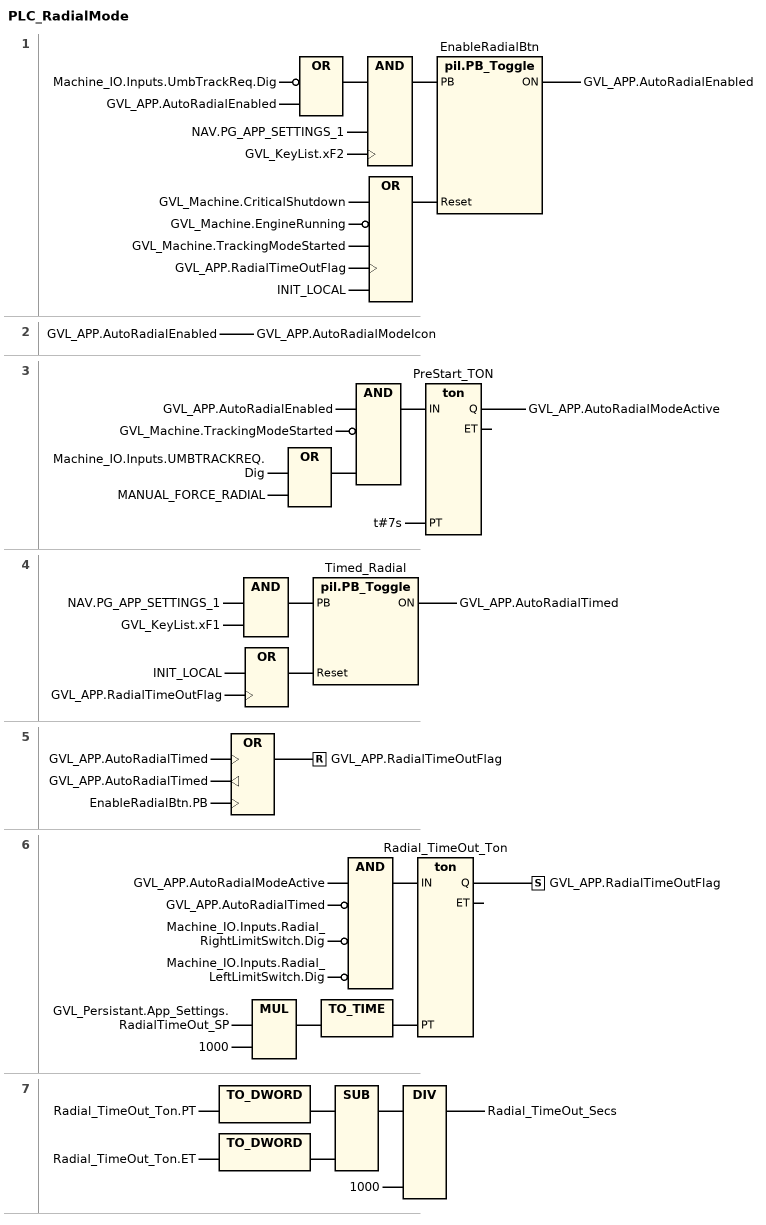
// NETWORK 1
_rt1(CLK := GVL_KeyList.xF2);
_rt2(CLK := GVL_APP.RadialTimeOutFlag);
EnableRadialBtn(PB := (NOT Machine_IO.Inputs.UmbTrackReq.Dig OR GVL_APP.AutoRadialEnabled) AND NAV.PG_APP_SETTINGS_1 AND _rt1.Q, Reset := GVL_Machine.CriticalShutdown OR NOT GVL_Machine.EngineRunning OR GVL_Machine.TrackingModeStarted OR _rt2.Q OR INIT_LOCAL); // pil.PB_Toggle
GVL_APP.AutoRadialEnabled := EnableRadialBtn.ON;

// NETWORK 2
GVL_APP.AutoRadialModeIcon := GVL_APP.AutoRadialEnabled;

// NETWORK 3
PreStart_TON(IN := GVL_APP.AutoRadialEnabled AND NOT GVL_Machine.TrackingModeStarted AND (Machine_IO.Inputs.UMBTRACKREQ.Dig OR MANUAL_FORCE_RADIAL), PT := t#7s); // ton
GVL_APP.AutoRadialModeActive := PreStart_TON.Q;

// NETWORK 4
_rt3(CLK := GVL_APP.RadialTimeOutFlag);
Timed_Radial(PB := NAV.PG_APP_SETTINGS_1 AND GVL_KeyList.xF1, Reset := INIT_LOCAL OR _rt3.Q); // pil.PB_Toggle
GVL_APP.AutoRadialTimed := Timed_Radial.ON;

// NETWORK 5
_rt4(CLK := GVL_APP.AutoRadialTimed);
_ft1(CLK := GVL_APP.AutoRadialTimed);
_rt5(CLK := EnableRadialBtn.PB);
GVL_APP.RadialTimeOutFlag R= _rt4.Q OR _ft1.Q OR _rt5.Q;

// NETWORK 6
Radial_TimeOut_Ton(IN := GVL_APP.AutoRadialModeActive AND NOT GVL_APP.AutoRadialTimed AND NOT Machine_IO.Inputs.Radial_RightLimitSwitch.Dig AND NOT Machine_IO.Inputs.Radial_LeftLimitSwitch.Dig, PT := TO_TIME(GVL_Persistant.App_Settings.RadialTimeOut_SP * 1000)); // ton
GVL_APP.RadialTimeOutFlag S= Radial_TimeOut_Ton.Q;

// NETWORK 7
Radial_TimeOut_Secs := (TO_DWORD(Radial_TimeOut_Ton.PT) - TO_DWORD(Radial_TimeOut_Ton.ET)) / 1000;

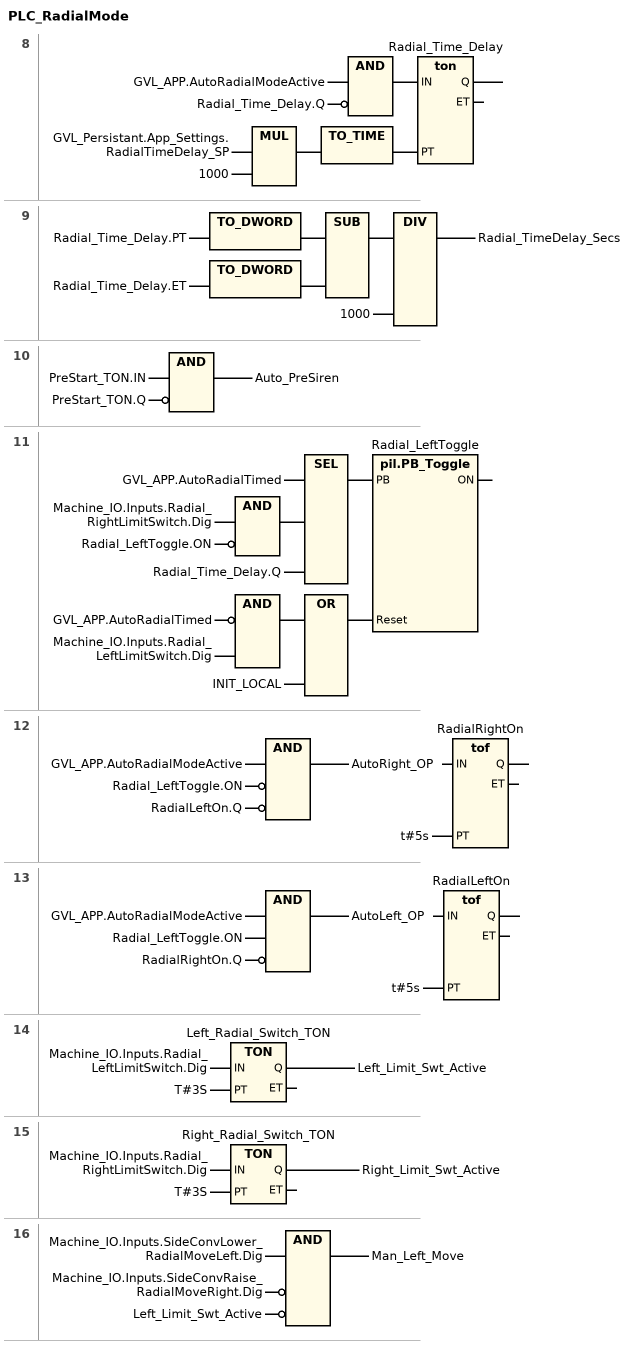
// NETWORK 8
Radial_Time_Delay(IN := GVL_APP.AutoRadialModeActive AND NOT Radial_Time_Delay.Q, PT := TO_TIME(GVL_Persistant.App_Settings.RadialTimeDelay_SP * 1000)); // ton

// NETWORK 9
Radial_TimeDelay_Secs := (TO_DWORD(Radial_Time_Delay.PT) - TO_DWORD(Radial_Time_Delay.ET)) / 1000;

// NETWORK 10
Auto_PreSiren := PreStart_TON.IN AND NOT PreStart_TON.Q;

// NETWORK 11
Radial_LeftToggle(PB := SEL(GVL_APP.AutoRadialTimed, Machine_IO.Inputs.Radial_RightLimitSwitch.Dig AND NOT Radial_LeftToggle.ON, Radial_Time_Delay.Q), Reset := NOT GVL_APP.AutoRadialTimed AND Machine_IO.Inputs.Radial_LeftLimitSwitch.Dig OR INIT_LOCAL); // pil.PB_Toggle

// NETWORK 12
_w1 := GVL_APP.AutoRadialModeActive AND NOT Radial_LeftToggle.ON AND NOT RadialLeftOn.Q;
AutoRight_OP := _w1;
RadialRightOn(IN := _w1, PT := t#5s); // tof

// NETWORK 13
_w2 := GVL_APP.AutoRadialModeActive AND Radial_LeftToggle.ON AND NOT RadialRightOn.Q;
AutoLeft_OP := _w2;
RadialLeftOn(IN := _w2, PT := t#5s); // tof

// NETWORK 14
Left_Radial_Switch_TON(IN := Machine_IO.Inputs.Radial_LeftLimitSwitch.Dig, PT := T#3S); // TON
Left_Limit_Swt_Active := Left_Radial_Switch_TON.Q;

// NETWORK 15
Right_Radial_Switch_TON(IN := Machine_IO.Inputs.Radial_RightLimitSwitch.Dig, PT := T#3S); // TON
Right_Limit_Swt_Active := Right_Radial_Switch_TON.Q;

// NETWORK 16
Man_Left_Move := Machine_IO.Inputs.SideConvLower_RadialMoveLeft.Dig AND NOT Machine_IO.Inputs.SideConvRaise_RadialMoveRight.Dig AND NOT Left_Limit_Swt_Active;

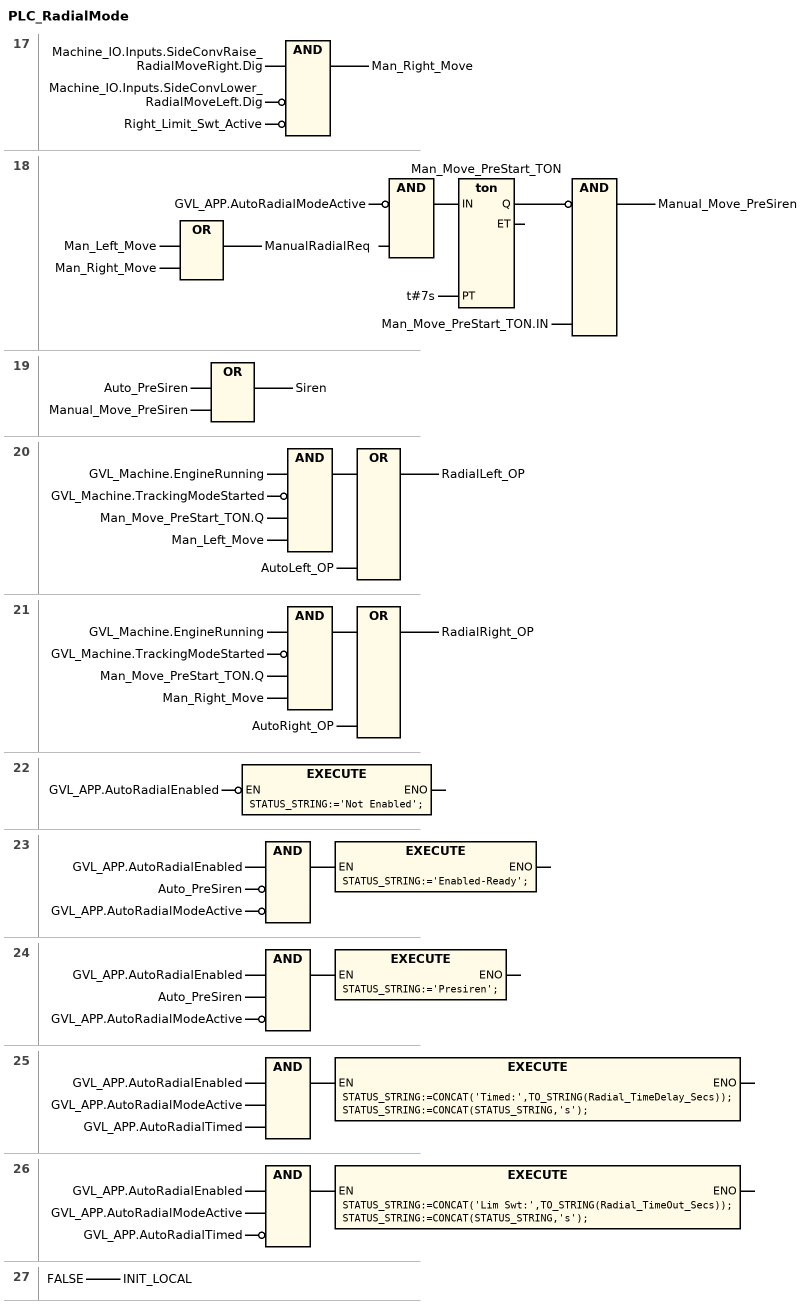
// NETWORK 17
Man_Right_Move := Machine_IO.Inputs.SideConvRaise_RadialMoveRight.Dig AND NOT Machine_IO.Inputs.SideConvLower_RadialMoveLeft.Dig AND NOT Right_Limit_Swt_Active;

// NETWORK 18
_w3 := Man_Left_Move OR Man_Right_Move;
ManualRadialReq := _w3;
Man_Move_PreStart_TON(IN := NOT GVL_APP.AutoRadialModeActive AND _w3, PT := t#7s); // ton
Manual_Move_PreSiren := NOT Man_Move_PreStart_TON.Q AND Man_Move_PreStart_TON.IN;

// NETWORK 19
Siren := Auto_PreSiren OR Manual_Move_PreSiren;

// NETWORK 20
RadialLeft_OP := GVL_Machine.EngineRunning AND NOT GVL_Machine.TrackingModeStarted AND Man_Move_PreStart_TON.Q AND Man_Left_Move OR AutoLeft_OP;

// NETWORK 21
RadialRight_OP := GVL_Machine.EngineRunning AND NOT GVL_Machine.TrackingModeStarted AND Man_Move_PreStart_TON.Q AND Man_Right_Move OR AutoRight_OP;

// NETWORK 22
IF NOT GVL_APP.AutoRadialEnabled THEN STATUS_STRING:='Not Enabled'; END_IF

// NETWORK 23
IF GVL_APP.AutoRadialEnabled AND NOT Auto_PreSiren AND NOT GVL_APP.AutoRadialModeActive THEN
    STATUS_STRING:='Enabled-Ready';
END_IF

// NETWORK 24
IF GVL_APP.AutoRadialEnabled AND Auto_PreSiren AND NOT GVL_APP.AutoRadialModeActive THEN
    STATUS_STRING:='Presiren';
END_IF

// NETWORK 25
IF GVL_APP.AutoRadialEnabled AND GVL_APP.AutoRadialModeActive AND GVL_APP.AutoRadialTimed THEN
    STATUS_STRING:=CONCAT('Timed:',TO_STRING(Radial_TimeDelay_Secs));
    STATUS_STRING:=CONCAT(STATUS_STRING,'s');
END_IF

// NETWORK 26
IF GVL_APP.AutoRadialEnabled AND GVL_APP.AutoRadialModeActive AND NOT GVL_APP.AutoRadialTimed THEN
    STATUS_STRING:=CONCAT('Lim Swt:',TO_STRING(Radial_TimeOut_Secs));
    STATUS_STRING:=CONCAT(STATUS_STRING,'s');
END_IF

// NETWORK 27
INIT_LOCAL := FALSE;

END_PROGRAM

// Device/Application/App_PLC/Control/PLC_JackLegs_SideConv
PROGRAM PLC_JackLegs_SideConv
VAR
	Prestart_TON: TON;
	Enable: BOOL;
	Siren: BOOL;
	Man_Side_Conv_Raise: BOOL;
	Man_Side_Conv_Lower: BOOL;
	Man_LHS_JackLegRaise: BOOL;
	Man_LHS_JackLegLower: BOOL;
	Man_RHS_JackLegRaise: BOOL;
	Man_RHS_JackLegLower: BOOL;
END_VAR
VAR // added by the converter: edge detectors and wires of the graphical bodies
    _w1 : BOOL;
END_VAR

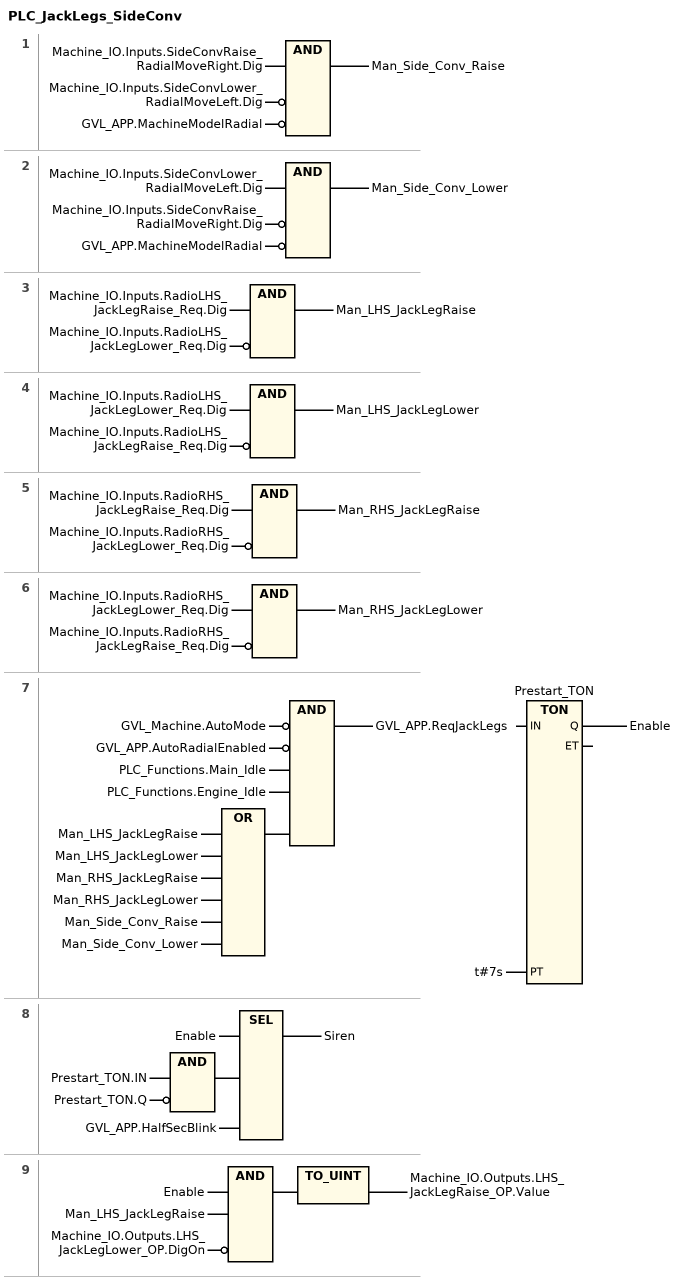
// NETWORK 1
Man_Side_Conv_Raise := Machine_IO.Inputs.SideConvRaise_RadialMoveRight.Dig AND NOT Machine_IO.Inputs.SideConvLower_RadialMoveLeft.Dig AND NOT GVL_APP.MachineModelRadial;

// NETWORK 2
Man_Side_Conv_Lower := Machine_IO.Inputs.SideConvLower_RadialMoveLeft.Dig AND NOT Machine_IO.Inputs.SideConvRaise_RadialMoveRight.Dig AND NOT GVL_APP.MachineModelRadial;

// NETWORK 3
Man_LHS_JackLegRaise := Machine_IO.Inputs.RadioLHS_JackLegRaise_Req.Dig AND NOT Machine_IO.Inputs.RadioLHS_JackLegLower_Req.Dig;

// NETWORK 4
Man_LHS_JackLegLower := Machine_IO.Inputs.RadioLHS_JackLegLower_Req.Dig AND NOT Machine_IO.Inputs.RadioLHS_JackLegRaise_Req.Dig;

// NETWORK 5
Man_RHS_JackLegRaise := Machine_IO.Inputs.RadioRHS_JackLegRaise_Req.Dig AND NOT Machine_IO.Inputs.RadioRHS_JackLegLower_Req.Dig;

// NETWORK 6
Man_RHS_JackLegLower := Machine_IO.Inputs.RadioRHS_JackLegLower_Req.Dig AND NOT Machine_IO.Inputs.RadioRHS_JackLegRaise_Req.Dig;

// NETWORK 7
_w1 := NOT GVL_Machine.AutoMode AND NOT GVL_APP.AutoRadialEnabled AND PLC_Functions.Main_Idle AND PLC_Functions.Engine_Idle AND (Man_LHS_JackLegRaise OR Man_LHS_JackLegLower OR Man_RHS_JackLegRaise OR Man_RHS_JackLegLower OR Man_Side_Conv_Raise OR Man_Side_Conv_Lower);
GVL_APP.ReqJackLegs := _w1;
Prestart_TON(IN := _w1, PT := t#7s); // TON
Enable := Prestart_TON.Q;

// NETWORK 8
Siren := SEL(Enable, Prestart_TON.IN AND NOT Prestart_TON.Q, GVL_APP.HalfSecBlink);

// NETWORK 9
Machine_IO.Outputs.LHS_JackLegRaise_OP.Value := TO_UINT(Enable AND Man_LHS_JackLegRaise AND NOT Machine_IO.Outputs.LHS_JackLegLower_OP.DigOn);

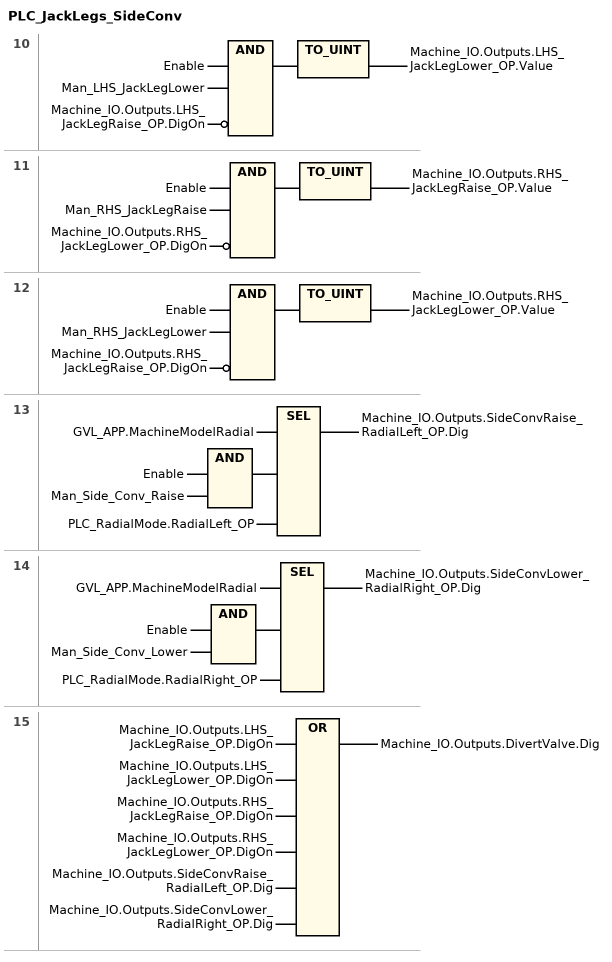
// NETWORK 10
Machine_IO.Outputs.LHS_JackLegLower_OP.Value := TO_UINT(Enable AND Man_LHS_JackLegLower AND NOT Machine_IO.Outputs.LHS_JackLegRaise_OP.DigOn);

// NETWORK 11
Machine_IO.Outputs.RHS_JackLegRaise_OP.Value := TO_UINT(Enable AND Man_RHS_JackLegRaise AND NOT Machine_IO.Outputs.RHS_JackLegLower_OP.DigOn);

// NETWORK 12
Machine_IO.Outputs.RHS_JackLegLower_OP.Value := TO_UINT(Enable AND Man_RHS_JackLegLower AND NOT Machine_IO.Outputs.RHS_JackLegRaise_OP.DigOn);

// NETWORK 13
Machine_IO.Outputs.SideConvRaise_RadialLeft_OP.Dig := SEL(GVL_APP.MachineModelRadial, Enable AND Man_Side_Conv_Raise, PLC_RadialMode.RadialLeft_OP);

// NETWORK 14
Machine_IO.Outputs.SideConvLower_RadialRight_OP.Dig := SEL(GVL_APP.MachineModelRadial, Enable AND Man_Side_Conv_Lower, PLC_RadialMode.RadialRight_OP);

// NETWORK 15
Machine_IO.Outputs.DivertValve.Dig := Machine_IO.Outputs.LHS_JackLegRaise_OP.DigOn OR Machine_IO.Outputs.LHS_JackLegLower_OP.DigOn OR Machine_IO.Outputs.RHS_JackLegRaise_OP.DigOn OR Machine_IO.Outputs.RHS_JackLegLower_OP.DigOn OR Machine_IO.Outputs.SideConvRaise_RadialLeft_OP.Dig OR Machine_IO.Outputs.SideConvLower_RadialRight_OP.Dig;

END_PROGRAM

// Device/Application/App_PLC/PLC_FanCtrl
PROGRAM PLC_FanCtrl
VAR
	OneSecTon: TON;
	Step: BYTE;
	WaitTon1: TON;
	WaitTon2: TON;

	RevTime_sec: WORD;
	THERMOSTAT: BOOL;
	//Fan_Forward_Time_Secs: UINT;
	STATUS_STRING: STRING;
	Forward_Time_Remaining: DWORD;
	Reverse_Time_Remaining: DWORD;
	Current_Forward_Time_STR: STRING;
END_VAR

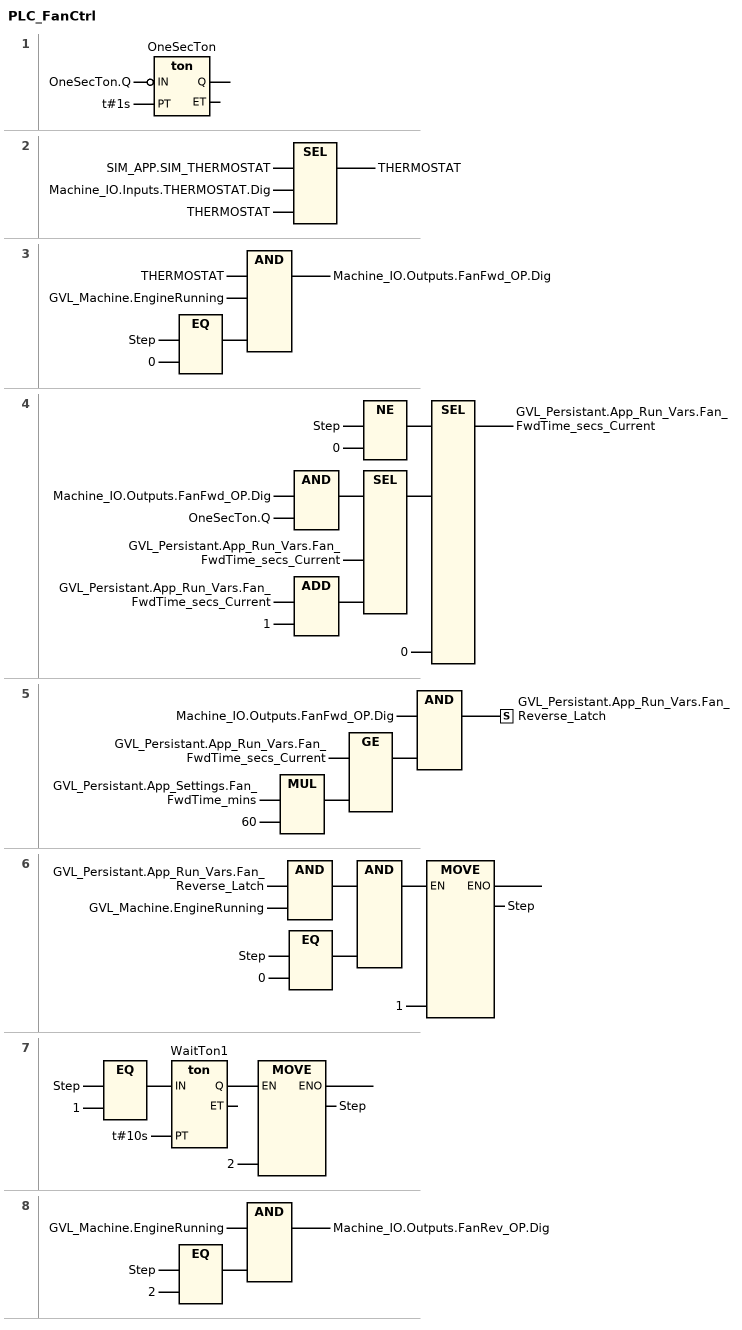
// NETWORK 1
OneSecTon(IN := NOT OneSecTon.Q, PT := t#1s); // ton

// NETWORK 2
THERMOSTAT := SEL(SIM_APP.SIM_THERMOSTAT, Machine_IO.Inputs.THERMOSTAT.Dig, THERMOSTAT);

// NETWORK 3
Machine_IO.Outputs.FanFwd_OP.Dig := THERMOSTAT AND GVL_Machine.EngineRunning AND Step = 0;

// NETWORK 4
GVL_Persistant.App_Run_Vars.Fan_FwdTime_secs_Current := SEL(Step <> 0, SEL(Machine_IO.Outputs.FanFwd_OP.Dig AND OneSecTon.Q, GVL_Persistant.App_Run_Vars.Fan_FwdTime_secs_Current, GVL_Persistant.App_Run_Vars.Fan_FwdTime_secs_Current + 1), 0);

// NETWORK 5
GVL_Persistant.App_Run_Vars.Fan_Reverse_Latch S= Machine_IO.Outputs.FanFwd_OP.Dig AND GVL_Persistant.App_Run_Vars.Fan_FwdTime_secs_Current >= GVL_Persistant.App_Settings.Fan_FwdTime_mins * 60;

// NETWORK 6
IF (GVL_Persistant.App_Run_Vars.Fan_Reverse_Latch AND GVL_Machine.EngineRunning) AND Step = 0 THEN
    Step := 1;
END_IF

// NETWORK 7
WaitTon1(IN := Step = 1, PT := t#10s); // ton
IF WaitTon1.Q THEN Step := 2; END_IF

// NETWORK 8
Machine_IO.Outputs.FanRev_OP.Dig := GVL_Machine.EngineRunning AND Step = 2;

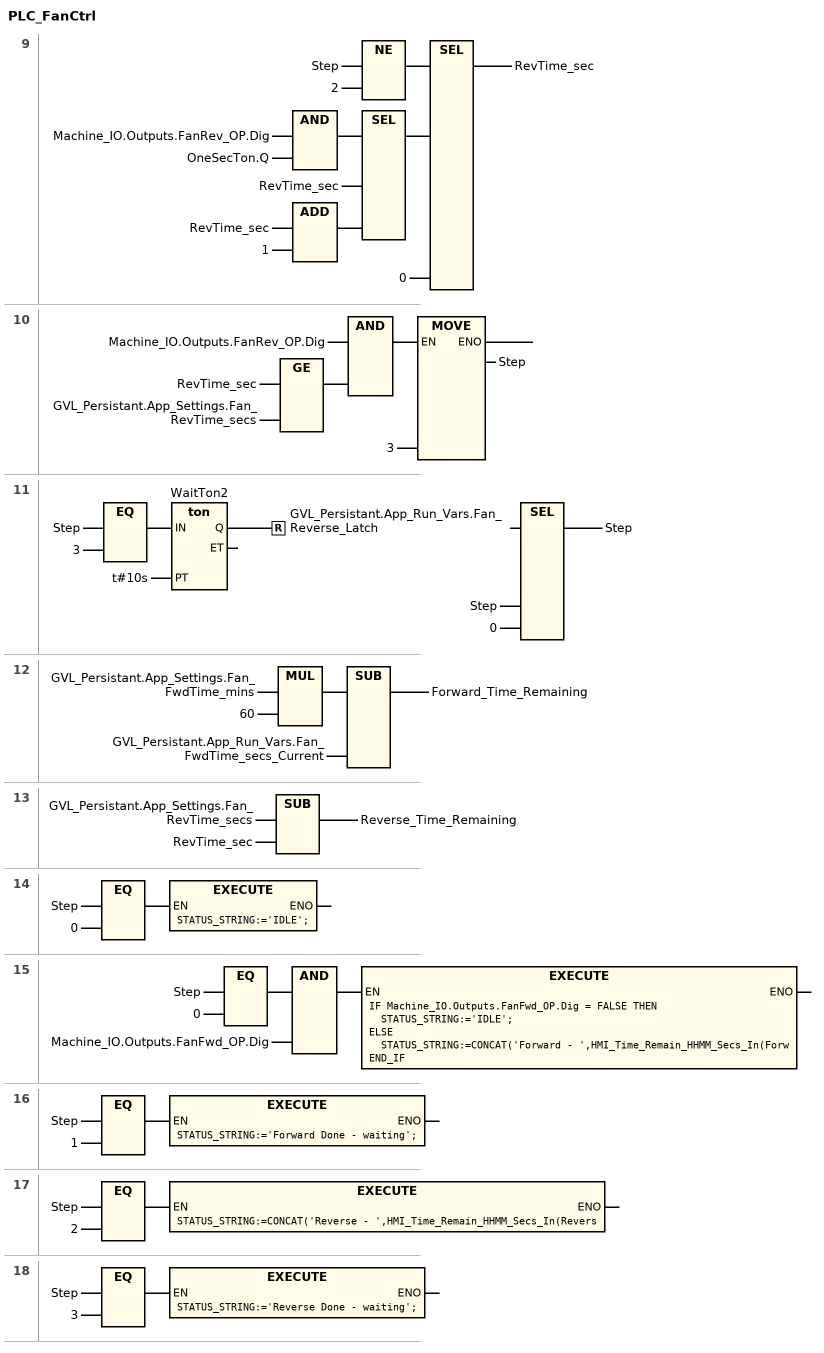
// NETWORK 9
RevTime_sec := SEL(Step <> 2, SEL(Machine_IO.Outputs.FanRev_OP.Dig AND OneSecTon.Q, RevTime_sec, RevTime_sec + 1), 0);

// NETWORK 10
IF Machine_IO.Outputs.FanRev_OP.Dig AND RevTime_sec >= GVL_Persistant.App_Settings.Fan_RevTime_secs THEN
    Step := 3;
END_IF

// NETWORK 11
WaitTon2(IN := Step = 3, PT := t#10s); // ton
GVL_Persistant.App_Run_Vars.Fan_Reverse_Latch R= WaitTon2.Q;
Step := SEL(WaitTon2.Q, Step, 0);

// NETWORK 12
Forward_Time_Remaining := GVL_Persistant.App_Settings.Fan_FwdTime_mins * 60 - GVL_Persistant.App_Run_Vars.Fan_FwdTime_secs_Current;

// NETWORK 13
Reverse_Time_Remaining := GVL_Persistant.App_Settings.Fan_RevTime_secs - RevTime_sec;

// NETWORK 14
IF Step = 0 THEN STATUS_STRING:='IDLE'; END_IF

// NETWORK 15
IF Step = 0 AND Machine_IO.Outputs.FanFwd_OP.Dig THEN
    IF Machine_IO.Outputs.FanFwd_OP.Dig = FALSE THEN
    	STATUS_STRING:='IDLE';
    ELSE
    	STATUS_STRING:=CONCAT('Forward - ',HMI_Time_Remain_HHMM_Secs_In(Forward_Time_Remaining));	
    END_IF
END_IF

// NETWORK 16
IF Step = 1 THEN STATUS_STRING:='Forward Done - waiting'; END_IF

// NETWORK 17
IF Step = 2 THEN STATUS_STRING:=CONCAT('Reverse - ',HMI_Time_Remain_HHMM_Secs_In(Reverse_Time_Remaining)); END_IF

// NETWORK 18
IF Step = 3 THEN STATUS_STRING:='Reverse Done - waiting'; END_IF

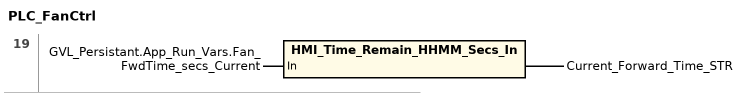
// NETWORK 19
Current_Forward_Time_STR := HMI_Time_Remain_HHMM_Secs_In(In := GVL_Persistant.App_Run_Vars.Fan_FwdTime_secs_Current);

END_PROGRAM

// Device/Application/App_PLC/CAN Comms/Engine Comms/HMI_Time_Remain_HHMM_Secs_In
FUNCTION HMI_Time_Remain_HHMM_Secs_In : STRING
VAR_INPUT
	In:DWORD;
END_VAR
VAR
	TotalSeconds: DWORD;
	Hours: DWORD;
	Mins: DWORD;
	Secs: DWORD;
	
	Temp_STR:STRING;
	TotalMinutes: DWORD;
END_VAR

TotalSeconds:=TO_DWORD(In);

TotalMinutes:=(TotalSeconds MOD (24*60*60))/60;

Hours:=TotalSeconds/(60*60);
Mins:=(TotalSeconds MOD (60*60))/60;
Secs:=TotalSeconds MOD 60;

Temp_STR:= '';

Temp_STR:= CONCAT(Temp_STR,DWORD_TO_STRING(Hours));
IF Hours < 10 THEN
	Temp_STR:= CONCAT(Temp_STR,'0');
END_IF

Temp_STR:= CONCAT(Temp_STR,':');

IF Mins < 10 THEN
	Temp_STR:= CONCAT(Temp_STR,'0');
END_IF
Temp_STR:= CONCAT(Temp_STR,DWORD_TO_STRING(Mins));

Temp_STR:= CONCAT(Temp_STR,':');

IF Secs < 10 THEN
	Temp_STR:= CONCAT(Temp_STR,'0');
END_IF
Temp_STR:= CONCAT(Temp_STR,DWORD_TO_STRING(Secs));


HMI_Time_Remain_HHMM_Secs_In := Temp_STR;

END_FUNCTION

// Device/Application/App_PLC/PLC_EngineRun
PROGRAM PLC_EngineRun
VAR
	TestBit1: BOOL;
	TempWord: WORD;
	TOF_0: tof;

	PreSirenTrig: BOOL;
	PreSirenTon: ton;
	PreSiren: BOOL;
	
	FastBlinkWait: ton;
	FastCountBlink: blink;
	FastBlinkTrig: R_trig;
	EngineSpeedPos_Count: SP_Count_VAR;
	
	WaitTon1: ton;
	WaitTof1: tof;

	TON_0: ton;
	BLINK_0: blink;
	PwrUpReset: BOOL;
	ECU_ENABLE: BOOL;
	SR_Auto_Stopped: SR;
END_VAR
VAR // added by the converter: edge detectors and wires of the graphical bodies
    _w1 : BOOL;
    _rt1, _rt2, _rt3 : R_TRIG;
    _ft1 : F_TRIG;
END_VAR

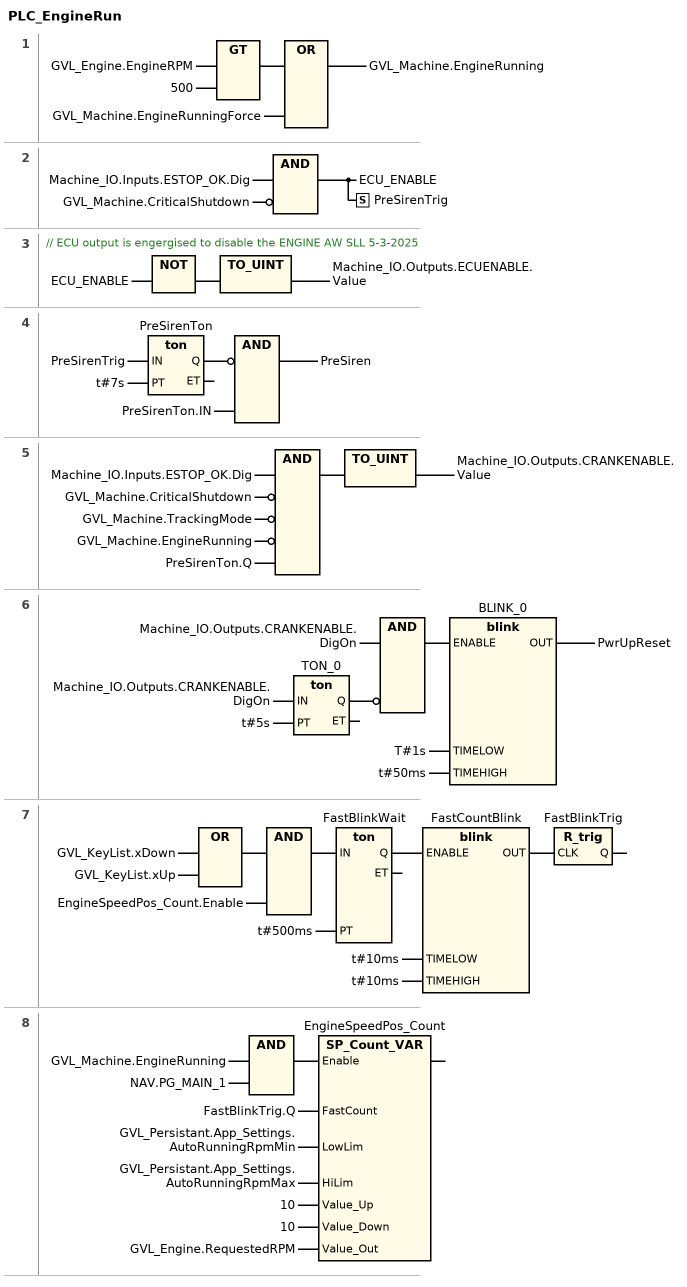
// NETWORK 1
GVL_Machine.EngineRunning := GVL_Engine.EngineRPM > 500 OR GVL_Machine.EngineRunningForce;

// NETWORK 2
_w1 := Machine_IO.Inputs.ESTOP_OK.Dig AND NOT GVL_Machine.CriticalShutdown;
ECU_ENABLE := _w1;
PreSirenTrig S= _w1;

// NETWORK 3
// // ECU output is engergised to disable the ENGINE AW SLL 5-3-2025
Machine_IO.Outputs.ECUENABLE.Value := TO_UINT(NOT ECU_ENABLE);

// NETWORK 4
PreSirenTon(IN := PreSirenTrig, PT := t#7s); // ton
PreSiren := NOT PreSirenTon.Q AND PreSirenTon.IN;

// NETWORK 5
Machine_IO.Outputs.CRANKENABLE.Value := TO_UINT(Machine_IO.Inputs.ESTOP_OK.Dig AND NOT GVL_Machine.CriticalShutdown AND NOT GVL_Machine.TrackingMode AND NOT GVL_Machine.EngineRunning AND PreSirenTon.Q);

// NETWORK 6
TON_0(IN := Machine_IO.Outputs.CRANKENABLE.DigOn, PT := t#5s); // ton
BLINK_0(ENABLE := Machine_IO.Outputs.CRANKENABLE.DigOn AND NOT TON_0.Q, TIMELOW := T#1s, TIMEHIGH := t#50ms); // blink
PwrUpReset := BLINK_0.OUT;

// NETWORK 7
FastBlinkWait(IN := (GVL_KeyList.xDown OR GVL_KeyList.xUp) AND EngineSpeedPos_Count.Enable, PT := t#500ms); // ton
FastCountBlink(ENABLE := FastBlinkWait.Q, TIMELOW := t#10ms, TIMEHIGH := t#10ms); // blink
FastBlinkTrig(CLK := FastCountBlink.OUT); // R_trig

// NETWORK 8
EngineSpeedPos_Count(
    Enable := GVL_Machine.EngineRunning AND NAV.PG_MAIN_1,
    FastCount := FastBlinkTrig.Q,
    LowLim := GVL_Persistant.App_Settings.AutoRunningRpmMin,
    HiLim := GVL_Persistant.App_Settings.AutoRunningRpmMax,
    Value_Up := 10,
    Value_Down := 10,
    Value_Out := GVL_Engine.RequestedRPM); // SP_Count_VAR

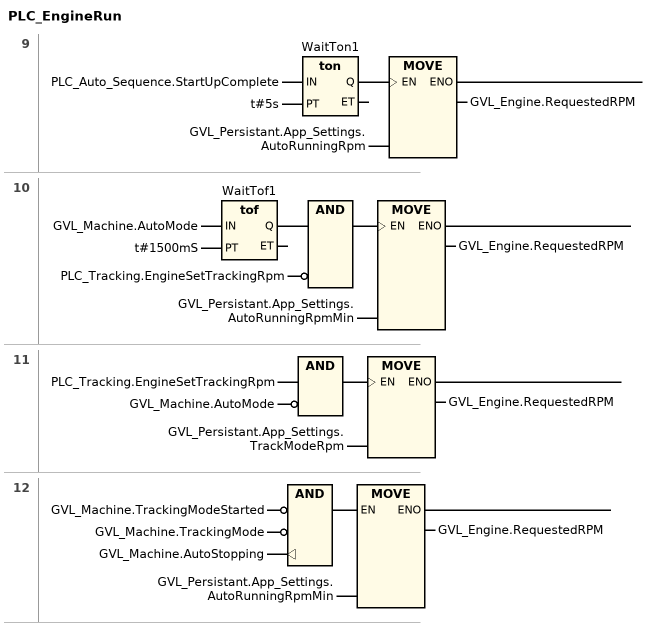
// NETWORK 9
WaitTon1(IN := PLC_Auto_Sequence.StartUpComplete, PT := t#5s); // ton
_rt1(CLK := WaitTon1.Q);
IF _rt1.Q THEN GVL_Engine.RequestedRPM := GVL_Persistant.App_Settings.AutoRunningRpm; END_IF

// NETWORK 10
WaitTof1(IN := GVL_Machine.AutoMode, PT := t#1500mS); // tof
_rt2(CLK := WaitTof1.Q AND NOT PLC_Tracking.EngineSetTrackingRpm);
IF _rt2.Q THEN GVL_Engine.RequestedRPM := GVL_Persistant.App_Settings.AutoRunningRpmMin; END_IF

// NETWORK 11
_rt3(CLK := PLC_Tracking.EngineSetTrackingRpm AND NOT GVL_Machine.AutoMode);
IF _rt3.Q THEN GVL_Engine.RequestedRPM := GVL_Persistant.App_Settings.TrackModeRpm; END_IF

// NETWORK 12
_ft1(CLK := GVL_Machine.AutoStopping);
IF NOT GVL_Machine.TrackingModeStarted AND NOT GVL_Machine.TrackingMode AND _ft1.Q THEN
    GVL_Engine.RequestedRPM := GVL_Persistant.App_Settings.AutoRunningRpmMin;
END_IF

END_PROGRAM

// Device/Application/App_PLC/Set Points/SP_Count_VAR
FUNCTION_BLOCK SP_Count_VAR
VAR_INPUT
	Enable: BOOL;
	FastCount: BOOL;
	LowLim: WORD;
	HiLim: WORD;
	Value_Up: WORD;
	Value_Down: WORD;
END_VAR
VAR_IN_OUT
	Value_Out: WORD;
END_VAR
VAR // added by the converter: edge detectors and wires of the graphical bodies
    _rt1, _rt2 : R_TRIG;
END_VAR

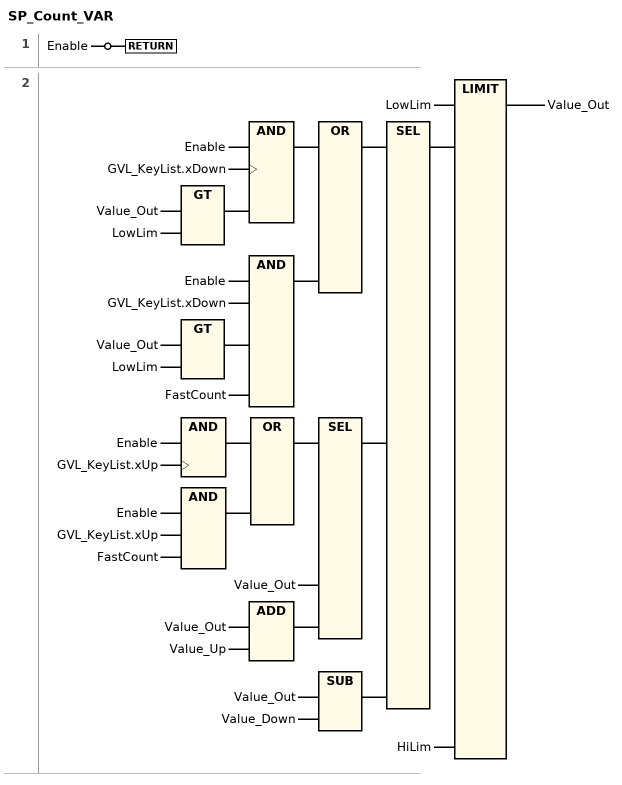
// NETWORK 1
IF NOT Enable THEN RETURN; END_IF

// NETWORK 2
_rt1(CLK := GVL_KeyList.xDown);
_rt2(CLK := GVL_KeyList.xUp);
Value_Out := LIMIT(LowLim, SEL(Enable AND _rt1.Q AND Value_Out > LowLim OR Enable AND GVL_KeyList.xDown AND Value_Out > LowLim AND FastCount, SEL(Enable AND _rt2.Q OR Enable AND GVL_KeyList.xUp AND FastCount, Value_Out, Value_Out + Value_Up), Value_Out - Value_Down), HiLim);

END_FUNCTION_BLOCK

// Device/Application/App_PLC/CAN Comms/CAN_TX_AUX_IO
  PROGRAM CAN_TX_AUX_IO
VAR
	EnableCAN0: ifmRCAN.CAN_Enable;
	Rx_200: ifmrcan.CAN_Rx;
	aUSINT_TO_aBYTE_200: PIL.aUSINT_TO_aBYTE;
	Rx200: ARRAY[0..7] OF USINT;	
	Tx201: ifmrcan.CAN_Tx;
	Tx201_Ton: TON;
	HEARTBEAT: BLINK;
	RX200_UNAVAIL_TON: TON;
	RX200_AVAIL_PULSE: BOOL;
	NODE_AUX_ALLOW_UNAVIL: BOOL := FALSE;
END_VAR
VAR // added by the converter: edge detectors and wires of the graphical bodies
    _w1 : BOOL;
END_VAR

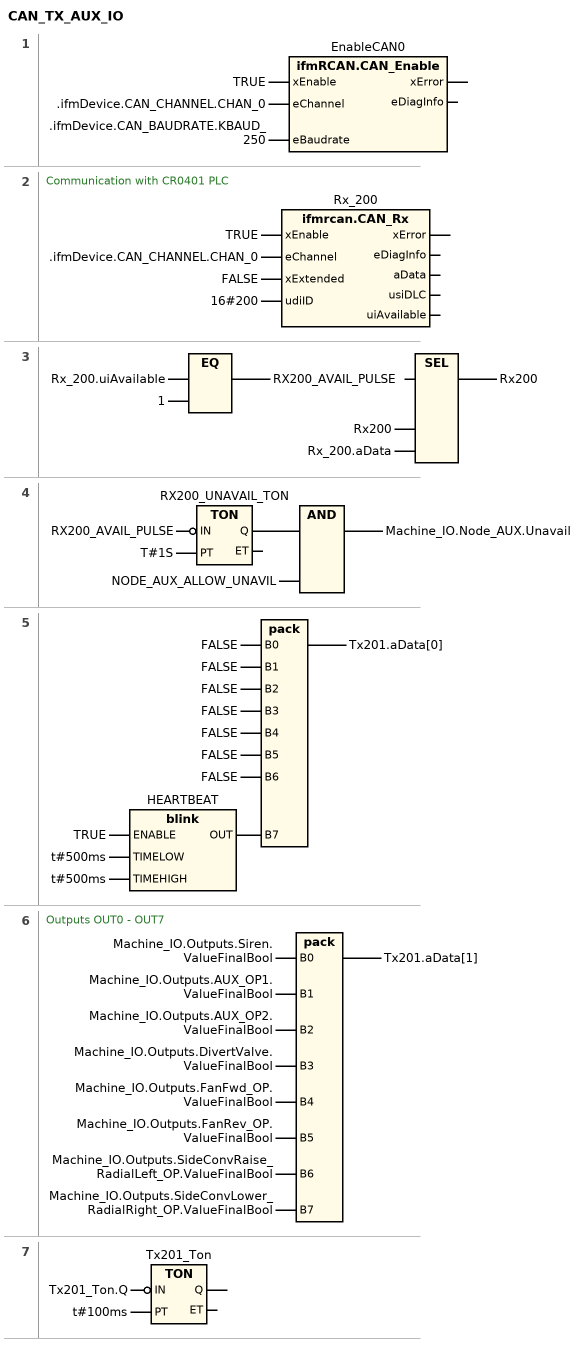
// NETWORK 1
EnableCAN0(
    xEnable := TRUE,
    eChannel := .ifmDevice.CAN_CHANNEL.CHAN_0,
    eBaudrate := .ifmDevice.CAN_BAUDRATE.KBAUD_250); // ifmRCAN.CAN_Enable

// NETWORK 2
// Communication with CR0401 PLC
Rx_200(xEnable := TRUE, eChannel := .ifmDevice.CAN_CHANNEL.CHAN_0, xExtended := FALSE, udiID := 16#200); // ifmrcan.CAN_Rx

// NETWORK 3
_w1 := Rx_200.uiAvailable = 1;
RX200_AVAIL_PULSE := _w1;
Rx200 := SEL(_w1, Rx200, Rx_200.aData);

// NETWORK 4
RX200_UNAVAIL_TON(IN := NOT RX200_AVAIL_PULSE, PT := T#1S); // TON
Machine_IO.Node_AUX.Unavail := RX200_UNAVAIL_TON.Q AND NODE_AUX_ALLOW_UNAVIL;

// NETWORK 5
HEARTBEAT(ENABLE := TRUE, TIMELOW := t#500ms, TIMEHIGH := t#500ms); // blink
Tx201.aData[0] := pack(B0 := FALSE, B1 := FALSE, B2 := FALSE, B3 := FALSE, B4 := FALSE, B5 := FALSE, B6 := FALSE, B7 := HEARTBEAT.OUT);

// NETWORK 6
// Outputs OUT0 - OUT7
Tx201.aData[1] := pack(B0 := Machine_IO.Outputs.Siren.ValueFinalBool, B1 := Machine_IO.Outputs.AUX_OP1.ValueFinalBool, B2 := Machine_IO.Outputs.AUX_OP2.ValueFinalBool, B3 := Machine_IO.Outputs.DivertValve.ValueFinalBool, B4 := Machine_IO.Outputs.FanFwd_OP.ValueFinalBool, B5 := Machine_IO.Outputs.FanRev_OP.ValueFinalBool, B6 := Machine_IO.Outputs.SideConvRaise_RadialLeft_OP.ValueFinalBool, B7 := Machine_IO.Outputs.SideConvLower_RadialRight_OP.ValueFinalBool);

// NETWORK 7
Tx201_Ton(IN := NOT Tx201_Ton.Q, PT := t#100ms); // TON

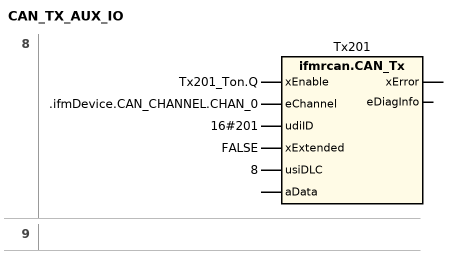
// NETWORK 8
Tx201(
    xEnable := Tx201_Ton.Q,
    eChannel := .ifmDevice.CAN_CHANNEL.CHAN_0,
    udiID := 16#201,
    xExtended := FALSE,
    usiDLC := 8); // ifmrcan.CAN_Tx

// NETWORK 9

END_PROGRAM

// Device/Application/App_Common/System/SECURITY_COM
PROGRAM SECURITY_COM
VAR
	INIT: BOOL := TRUE;
	PIN_CODE_ENTERED: LWORD;
	PIN_CODE_FIXED: LWORD:=1605;
END_VAR

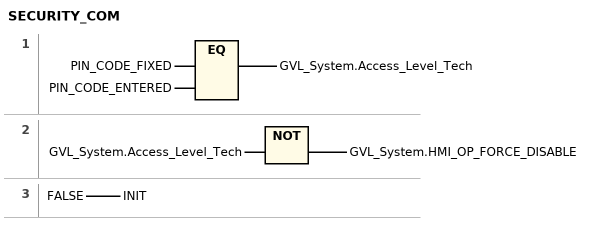
// NETWORK 1
GVL_System.Access_Level_Tech := PIN_CODE_FIXED = PIN_CODE_ENTERED;

// NETWORK 2
GVL_System.HMI_OP_FORCE_DISABLE := NOT GVL_System.Access_Level_Tech;

// NETWORK 3
INIT := FALSE;

END_PROGRAM

// Device/Application/App_Common/Alarms/Alarms_Task
PROGRAM Alarms_Task
VAR
END_VAR

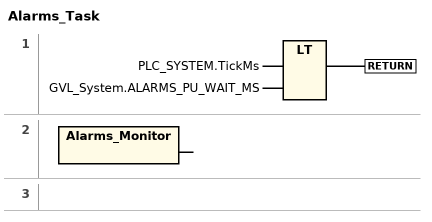
// NETWORK 1
IF PLC_SYSTEM.TickMs < GVL_System.ALARMS_PU_WAIT_MS THEN RETURN; END_IF

// NETWORK 2
Alarms_Monitor();

// NETWORK 3

END_PROGRAM

// Device/Application/App_Common/Alarms/Alarms_Monitor
PROGRAM Alarms_Monitor
VAR
	PRIME_ARRAY: BOOL;
END_VAR
VAR // added by the converter: edge detectors and wires of the graphical bodies
    _rt1 : R_TRIG;
END_VAR

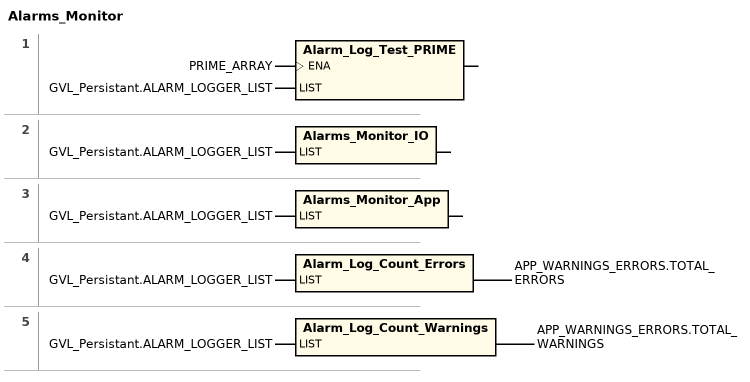
// NETWORK 1
_rt1(CLK := PRIME_ARRAY);
Alarm_Log_Test_PRIME(ENA := _rt1.Q, LIST := GVL_Persistant.ALARM_LOGGER_LIST);

// NETWORK 2
Alarms_Monitor_IO(LIST := GVL_Persistant.ALARM_LOGGER_LIST);

// NETWORK 3
Alarms_Monitor_App(LIST := GVL_Persistant.ALARM_LOGGER_LIST);

// NETWORK 4
APP_WARNINGS_ERRORS.TOTAL_ERRORS := Alarm_Log_Count_Errors(LIST := GVL_Persistant.ALARM_LOGGER_LIST);

// NETWORK 5
APP_WARNINGS_ERRORS.TOTAL_WARNINGS := Alarm_Log_Count_Warnings(LIST := GVL_Persistant.ALARM_LOGGER_LIST);

END_PROGRAM

// Device/Application/LIBS/Alarms/Functions/Alarm_Log_Test_PRIME
FUNCTION Alarm_Log_Test_PRIME : INT
VAR_INPUT
	ENA: BOOL;
	LIST: REFERENCE TO SLL_LOGGER_MAIN_SRUCT;
END_VAR
VAR_OUTPUT
END_VAR
VAR
	Empty: SLL_LOGGER_ITEM;
	X:WORD;
	Result : RTS_IEC_RESULT;	
	TimestampTemp:SYSTIME;
END_VAR

IF ENA = FALSE THEN
	RETURN;
END_IF

FOR X := 0 TO (LIST.LOGGER_LIST_SIZE-1) DO
	Result := SysTimeRtcHighResGet(TimestampTemp);
	LIST.LOGGER_LIST[X].Empty:=FALSE;
	LIST.LOGGER_LIST[X].ID:=X+9000;
	LIST.LOGGER_LIST[X].TimeDateTriggered:=TimestampTemp;
	LIST.LOGGER_LIST[X].Addtional_Info := CONCAT('Add_Info: ',TO_STRING(X));
	LIST.LOGGER_LIST[X].Flags.Active:=TRUE;
	LIST.LOGGER_LIST[X].Group.ErrorApp:=TRUE;	
END_FOR

END_FUNCTION

// Device/Application/App_CODE_GEN/MAIN_CODE_GEN/App_CODE_GEN/Alarms/Alarms_Monitor_IO
PROGRAM Alarms_Monitor_IO
VAR_INPUT
	LIST: REFERENCE TO SLL_LOGGER_MAIN_SRUCT;	
END_VAR
VAR
	IO_Error_Group: SLL_LOGGER_ITEM_GROUP:=(ErrorIO:=1);

// Alarms_Monitor_IO_Declare_CODE_GEN_START

// generated (UTC): 2024-07-23 18:31:25.297397+00:00

	ESTOPS_SAFETY_RELAY: SLL_AlarmBit;
	OVERRIDE_GENERAL_SWT: SLL_AlarmBit;
	FUNCTIONS_DEADMAN_CHASSIS_BTN: SLL_AlarmBit;
	CABIN_RAISE_CHASSIS_BTN: SLL_AlarmBit;
	CABIN_LOWER_CHASSIS_BTN: SLL_AlarmBit;
	JACKLEGS_DOWN_CHASSIS_BTN: SLL_AlarmBit;
	JACKLEGS_UP_CHASSIS_BTN: SLL_AlarmBit;
	ENGINE_START_CHASSIS_BTN: SLL_AlarmBit;
	HYDRAULICS_DC_PUMP_RUNNING_SIG: SLL_AlarmBit;
	JACKLEGS_STOWED_DOWN_PRESSURE_SWT: SLL_AlarmBit;
	JACKLEGS_STOWED_UP_PRESSURE_SWT: SLL_AlarmBit;
	MAINS_AC_MAINS_CONNECTED: SLL_AlarmBit;
	TRUCK_NEUTRAL_FROM_TRUCK : SLL_AlarmBit;
	SPARE_CHASSIS_IN0701: SLL_AlarmBit;
	CABIN_PART_RAISED_DIG: SLL_AlarmBit;
	SPARE_CHASSIS_IN0703: SLL_AlarmBit;
	CABIN_LOWER_LIMIT_DIG: SLL_AlarmBit;
	CABIN_FULLY_STOWED_DIG: SLL_AlarmBit;
	PTO_ACTIVE_SIG: SLL_AlarmBit;
	FUNCTIONS_CHASSIS_CABIN_CHANGE_OVER_SWT: SLL_AlarmBit;
	LIGHTS_SIDE_LIGHTS_DASH_SIG: SLL_AlarmBit;
	TRUCK_HANDBRAKE_APPLIED_SIGNAL: SLL_AlarmBit;
	ENGINE_RUNNING_SIGNAL: SLL_AlarmBit;
	TRUCK_REVERSE_FROM_TRUCK: SLL_AlarmBit;
	SPARE_CHASSIS_IN0400: SLL_AlarmBit;
	ENGINE_STOP_CHASSIS_BTN: SLL_AlarmBit;
	HYDRAULICS_OIL_LEVEL_RES: SLL_AlarmBit;
	SPARE_CHASSIS_IN0901: SLL_AlarmBit;
	SPARE_CHASSIS_IN0300: SLL_AlarmBit;
	SPARE_CHASSIS_IN0301: SLL_AlarmBit;
	JACKLEGS_CYCLINDER_100_BAR_PRESSURE_SWT: SLL_AlarmBit;
	JACKLEGS_CYCLINDER_150_BAR_PRESSURE_SWT: SLL_AlarmBit;
	ENGINE_STOP_COMMAND: SLL_AlarmBit;
	CHASSIS_SIREN: SLL_AlarmBit;
	SPARE_CHASSIS_OUT0002: SLL_AlarmBit;
	JACKLEGS_WARNING_BEACON: SLL_AlarmBit;
	HYDRAULICS_OIL_LEVEL_WARNING_LED: SLL_AlarmBit;
	SPARE_CHASSIS_OUT0005: SLL_AlarmBit;
	HYDRAULICS_MASTER_VALVE: SLL_AlarmBit;
	PTO_TOGGLE: SLL_AlarmBit;
	SPARE_CHASSIS_OUT0008: SLL_AlarmBit;
	CHASSIS_Supply_GROUP0: SLL_AlarmBit;
	SPARE_CHASSIS_OUT0100: SLL_AlarmBit;
	ENGINE_START_COMMAND: SLL_AlarmBit;
	SPARE_CHASSIS_OUT0102: SLL_AlarmBit;
	PLATFORM_TRAVERSE_LEFT_VALVE: SLL_AlarmBit;
	SPARE_CHASSIS_OUT0104: SLL_AlarmBit;
	CABIN_RAISE_COMMAND: SLL_AlarmBit;
	CABIN_LOWER_COMMAND: SLL_AlarmBit;
	JACKLEGS_UP_COMMAND: SLL_AlarmBit;
	JACKLEGS_DOWN_COMMAND: SLL_AlarmBit;
	CHASSIS_Supply_GROUP1: SLL_AlarmBit;
	HYDRAULICS_MASTER_LED_CAB: SLL_AlarmBit;
	OVERRIDE_DRIVE_INTERLOCK_ACTIVE_LED: SLL_AlarmBit;
	CABIN_FULLY_STOWED_LED: SLL_AlarmBit;
	JACKLEGS_STOWED_LED: SLL_AlarmBit;
	JACKLEGS_DOWN_LED: SLL_AlarmBit;
	CABIN_RAISED_LED: SLL_AlarmBit;
	PLATFORM_TRAVERSE_RIGHT_VALVE: SLL_AlarmBit;
	PLATFORM_RETRACT_COMMAND: SLL_AlarmBit;
	PLATFORM_EXTEND_COMMAND: SLL_AlarmBit;
	CHASSIS_Supply_GROUP2: SLL_AlarmBit;
	SPARE_CHASSIS_OUT3000: SLL_AlarmBit;
	SPARE_CHASSIS_OUT3001: SLL_AlarmBit;
	SPARE_CABIN_IN0100: SLL_AlarmBit;
	PLATFORM_EXTEND_BTN: SLL_AlarmBit;
	PLATFORM_RETRACT_BTN: SLL_AlarmBit;
	PLATFORM_SIDERAILS_LHS_SIDERAILS_STOWED_DIG: SLL_AlarmBit;
	PLATFORM_SIDERAILS_RHS_SIDERAILS_STOWED_DIG: SLL_AlarmBit;
	PLATFORM_TRAVERSE_STOWED_DIG: SLL_AlarmBit;
	SPARE_CABIN_IN0202: SLL_AlarmBit;
	PLATFORM_LEUZE_SENSORS_LEFT_SENSOR_DIG: SLL_AlarmBit;
	PLATFORM_LEUZE_SENSORS_RIGHT_SENSOR_DIG: SLL_AlarmBit;
	PLATFORM_FULLY_STOWED_DIG: SLL_AlarmBit;
	PLATFORM_PART_STOWED_DIG: SLL_AlarmBit;
	DOORS_REAR_DOOR_CLOSED_SIG: SLL_AlarmBit;
	PLATFORM_SAFETY_GATES_LHS_EDGE_SENSOR: SLL_AlarmBit;
	SPARE_CABIN_IN0701: SLL_AlarmBit;
	SPARE_CABIN_IN0702: SLL_AlarmBit;
	PLATFORM_SAFETY_GATES_RHS_EDGE_SENSOR: SLL_AlarmBit;
	SPARE_CABIN_IN0000: SLL_AlarmBit;
	PLATFORM_SAFETY_GATES_LHS_GATE_CLOSED_SIGNAL: SLL_AlarmBit;
	PLATFORM_SAFETY_GATES_RHS_GATE_CLOSED_SIGNAL: SLL_AlarmBit;
	SPARE_CABIN_IN0003: SLL_AlarmBit;
	CAS_RESET_SWT: SLL_AlarmBit;
	CAS_TORTOISE_SWT: SLL_AlarmBit;
	CAS_ENABLE_ON_OFF_SWT: SLL_AlarmBit;
	SPARE_CABIN_IN0503: SLL_AlarmBit;
	PLATFORM_SAFETY_EDGE_SAFETY_BUMPER_RES_ANA: SLL_AlarmBit;
	SPARE_CABIN_IN0401: SLL_AlarmBit;
	PLATFORM_TRAVERSE_LEFT_BTN: SLL_AlarmBit;
	PLATFORM_TRAVERSE_RIGHT_BTN: SLL_AlarmBit;
	DOORS_SIDE_DOOR_CLOSED_SIG: SLL_AlarmBit;
	FUNCTIONS_DEADMAN_CABIN_BTN: SLL_AlarmBit;
	SPARE_CABIN_IN0800: SLL_AlarmBit;
	SPARE_CABIN_IN0801: SLL_AlarmBit;
	PLATFORM_SIDERAILS_SIDERAILS_STOWED_LED: SLL_AlarmBit;
	PLATFORM_SAFETY_GATES_UNLOCK_1: SLL_AlarmBit;
	TRUCK_FORCE_NEUTRAL: SLL_AlarmBit;
	PLATFORM_SAFETY_GATES_UNLOCK_2: SLL_AlarmBit;
	CAS_LOCKOUT_LED: SLL_AlarmBit;
	PLATFORM_EXTENDED_LED: SLL_AlarmBit;
	PLATFORM_RETRACTED_LED: SLL_AlarmBit;
	CAS_TORTOISE_MODE_LED: SLL_AlarmBit;
	CAS_DRIVERS_BUZZER: SLL_AlarmBit;
	CABIN_Supply_GROUP0: SLL_AlarmBit;
	DOORS_ALLOW_SIDE_DOOR: SLL_AlarmBit;
	DOORS_ALLOW_REAR_DOOR: SLL_AlarmBit;
	SPARE_CABIN_OUT0102: SLL_AlarmBit;
	SPARE_CABIN_OUT0103: SLL_AlarmBit;
	SPARE_CABIN_OUT0104: SLL_AlarmBit;
	SPARE_CABIN_OUT0105: SLL_AlarmBit;
	SPARE_CABIN_OUT0106: SLL_AlarmBit;
	SPARE_CABIN_OUT0107: SLL_AlarmBit;
	SPARE_CABIN_OUT0108: SLL_AlarmBit;
	CABIN_Supply_GROUP1: SLL_AlarmBit;
	SPARE_CABIN_OUT0200: SLL_AlarmBit;
	LIGHTS_LEFT_SIDE_LIGHTS: SLL_AlarmBit;
	CAS_GREEN_BEACON: SLL_AlarmBit;
	FUNCTIONS_DEADMAN_CABIN_BTN_LED: SLL_AlarmBit;
	SPARE_CABIN_OUT0204: SLL_AlarmBit;
	SPARE_CABIN_OUT0205: SLL_AlarmBit;
	LIGHTS_SIDE_RLY: SLL_AlarmBit;
	SPARE_CABIN_OUT0207: SLL_AlarmBit;
	SPARE_CABIN_OUT0208: SLL_AlarmBit;
	CABIN_Supply_GROUP2: SLL_AlarmBit;
	SPARE_CABIN_OUT3000: SLL_AlarmBit;
	SPARE_CABIN_OUT3001: SLL_AlarmBit;
	// Alarms_Monitor_IO_Declare_CODE_GEN_STOP	
END_VAR


// Alarms_Monitor_IO_STL_Body_CODE_GEN_START

// generated (UTC): 2024-07-23 18:31:25.307398+00:00

// Alarms_Monitor_IO_STL_Body_CODE_GEN_STOP

END_PROGRAM

// Device/Application/LIBS/Alarms/Functions/SLL_AlarmBit
FUNCTION_BLOCK SLL_AlarmBit
VAR_INPUT
	LIST: REFERENCE TO SLL_LOGGER_MAIN_SRUCT;
	ID:WORD;
	Bit_Input:BOOL;
	Description:STRING;
	Add_Info:STRING;
	Group: SLL_LOGGER_ITEM_GROUP;
	HushOption: BOOL:=FALSE;
END_VAR
VAR_OUTPUT
END_VAR
VAR
	Init: BOOL;
	Bit_Input_Prev:BOOL;
	
	HashCode:ULINT; // based on high resolution time and the ID!
END_VAR

IF Bit_Input_Prev <> Bit_Input THEN
	IF Bit_Input THEN
		HashCode:=Alarm_Log_Add(LIST,ID,Description,Add_Info,Group,HushOption);
	ELSE
		Alarm_Log_Update(LIST,Bit_Input,HashCode);
	END_IF
	Bit_Input_Prev := Bit_Input;
END_IF

END_FUNCTION_BLOCK

// Device/Application/LIBS/Alarms/Functions/Alarm_Log_Add
FUNCTION Alarm_Log_Add : ULINT
VAR_INPUT
	LIST: REFERENCE TO SLL_LOGGER_MAIN_SRUCT;
	ID: WORD; // base id of the alarm
	Description: STRING; // Additional information for the alarm
	Addtional_Info: STRING; // Additional information for the alarm
	Group: SLL_LOGGER_ITEM_GROUP;
	HushOption:BOOL;
END_VAR
VAR_OUTPUT
END_VAR
VAR
	X:WORD;
	Result : RTS_IEC_RESULT;	
	TimestampTemp:SYSTIME;
END_VAR

// shift down the aray - loose the oldest data
FOR X :=(LIST.LOGGER_LIST_SIZE-1) TO 1 BY -1 DO
	LIST.LOGGER_LIST[X]:=LIST.LOGGER_LIST[X-1];
END_FOR

Result := SysTimeRtcHighResGet(TimestampTemp);

LIST.LOGGER_LIST[0].Addtional_Info := Addtional_Info;

LIST.LOGGER_LIST[0].Flags.Active:=TRUE;
LIST.LOGGER_LIST[0].Flags.Acknowledged:=0;

LIST.LOGGER_LIST[0].Group:=Group;

LIST.LOGGER_LIST[0].ID:=ID;
LIST.LOGGER_LIST[0].TimeDateTriggered:=TimestampTemp;

LIST.LOGGER_LIST[0].Group.HushOption:=HushOption;

Alarm_Log_Add:=SHR(TimestampTemp,16);
Alarm_Log_Add:=Alarm_Log_Add OR TO_ULINT(ID);

END_FUNCTION

// Device/Application/LIBS/Alarms/Functions/Alarm_Log_Update
FUNCTION Alarm_Log_Update : INT
VAR_INPUT
	LIST: REFERENCE TO SLL_LOGGER_MAIN_SRUCT;	
	ActiveState:BOOL;
	HashCode: ULINT;
END_VAR
VAR_OUTPUT
END_VAR
VAR
	X:WORD;
	HashTemp:ULINT;
END_VAR

IF HashCode = 0 THEN
	RETURN; // aint note code!
END_IF

FOR X := 0 TO (LIST.LOGGER_LIST_SIZE-1) BY 1 DO	
	// go through each item in list
	IF LIST.LOGGER_LIST[X].ID > 0 THEN
		// got an id - generate the temp hash code
		HashTemp:=SHR(LIST.LOGGER_LIST[X].TimeDateTriggered,16);	
		HashTemp:=HashTemp OR TO_ULINT(LIST.LOGGER_LIST[X].ID);
		IF HashTemp = HashCode THEN
			// all matches - update the has code!
			LIST.LOGGER_LIST[X].Flags.Active:=ActiveState;
		END_IF		
	END_IF
END_FOR

END_FUNCTION

// Device/Application/App_CODE_GEN/MAIN_CODE_GEN/App_CODE_GEN/Alarms/Alarms_Monitor_App
PROGRAM Alarms_Monitor_App
VAR_INPUT
	LIST: REFERENCE TO SLL_LOGGER_MAIN_SRUCT;	
END_VAR
VAR
	App_Error_Group: SLL_LOGGER_ITEM_GROUP:=(ErrorApp:=1);	
	
// Alarms_Monitor_App_Declare_CODE_GEN_START

// generated (UTC): 2024-07-23 18:31:25.274396+00:00

	EMERGENCY_STOP_COMMON: SLL_AlarmBit;
	ETHERNET_PLC_COMMON_FAILURE: SLL_AlarmBit;
	ETHERNET_CHASSIS_PLC_MISSING: SLL_AlarmBit;
	ETHERNET_CHASSIS_PLC_ERROR_LT: SLL_AlarmBit;
	ETHERNET_CHASSIS_PLC_ERROR_DIFF: SLL_AlarmBit;
	ETHERNET_CHASSIS_PLC_ERROR_FROZEN: SLL_AlarmBit;
	ETHERNET_CHASSIS_PLC_WARNING_DIFF: SLL_AlarmBit;
	ETHERNET_CHASSIS_PLC_WARNING_FROZEN: SLL_AlarmBit;
	Battery_Voltage_Warning: SLL_AlarmBit;
	Hydraulic_Oil_Level_Low: SLL_AlarmBit;
	
	LowHydOilAlarm: SLL_AlarmBit; // 120
	HydTempAlarm: SLL_AlarmBit; // 121
	DrumHighPress_Alarm: SLL_AlarmBit; // 122
	LowFuelAlarm: SLL_AlarmBit;	// 123
	AutoShutdownAlarm: SLL_AlarmBit; // 124
	LowOilPressAlarm: SLL_AlarmBit; // 125
	EngineHiTempAlarm: SLL_AlarmBit; //126
	
	// Alarms_Monitor_App_Declare_CODE_GEN_STOP	
END_VAR


// Alarms_Monitor_App_STL_Body_CODE_GEN_START

// generated (UTC): 2024-07-23 18:31:25.284397+00:00

EMERGENCY_STOP_COMMON(LIST:=LIST,Bit_Input:=GVL_Alarms.EMERGENCY_STOP_COMMON,ID:=101,Add_Info:='',Group:=App_Error_Group,HushOption:=1);
ETHERNET_PLC_COMMON_FAILURE(LIST:=LIST,Bit_Input:=GVL_Alarms.ETHERNET_PLC_COMMON_FAILURE,ID:=102,Add_Info:='',Group:=App_Error_Group,HushOption:=0);
Battery_Voltage_Warning(LIST:=LIST,Bit_Input:=GVL_Alarms.Battery_Voltage_Warning,ID:=103,Add_Info:='',Group:=App_Error_Group,HushOption:=0);
LowHydOilAlarm(LIST:=LIST,Bit_Input:=GVL_Alarms.LowHydOilAlarm,ID:=104,Add_Info:='',Group:=App_Error_Group,HushOption:=0);
HydTempAlarm(LIST:=LIST,Bit_Input:=GVL_Alarms.HydTempAlarm,ID:=105,Add_Info:='',Group:=App_Error_Group,HushOption:=0);
DrumHighPress_Alarm(LIST:=LIST,Bit_Input:=GVL_Alarms.DrumHighPress_Alarm,ID:=106,Add_Info:='',Group:=App_Error_Group,HushOption:=0);
LowFuelAlarm(LIST:=LIST,Bit_Input:=GVL_Alarms.LowFuelAlarm,ID:=107,Add_Info:='',Group:=App_Error_Group,HushOption:=0);
AutoShutdownAlarm(LIST:=LIST,Bit_Input:=GVL_Alarms.AutoShutdownAlarm,ID:=108,Add_Info:='',Group:=App_Error_Group,HushOption:=0);
LowOilPressAlarm(LIST:=LIST,Bit_Input:=GVL_Alarms.LowOilPressAlarm,ID:=109,Add_Info:='',Group:=App_Error_Group,HushOption:=0);
EngineHiTempAlarm(LIST:=LIST,Bit_Input:=GVL_Alarms.EngineHiTempAlarm,ID:=110,Add_Info:='',Group:=App_Error_Group,HushOption:=0);

ETHERNET_CHASSIS_PLC_MISSING(LIST:=LIST,Bit_Input:=GVL_Alarms.ETHERNET_CHASSIS_PLC_MISSING,ID:=1100,Add_Info:='',Group:=App_Error_Group,HushOption:=0);
ETHERNET_CHASSIS_PLC_ERROR_LT(LIST:=LIST,Bit_Input:=GVL_Alarms.ETHERNET_CHASSIS_PLC_ERROR_LT,ID:=1101,Add_Info:='',Group:=App_Error_Group,HushOption:=0);
ETHERNET_CHASSIS_PLC_ERROR_DIFF(LIST:=LIST,Bit_Input:=GVL_Alarms.ETHERNET_CHASSIS_PLC_ERROR_DIFF,ID:=1102,Add_Info:='',Group:=App_Error_Group,HushOption:=0);
ETHERNET_CHASSIS_PLC_ERROR_FROZEN(LIST:=LIST,Bit_Input:=GVL_Alarms.ETHERNET_CHASSIS_PLC_ERROR_FROZEN,ID:=1103,Add_Info:='',Group:=App_Error_Group,HushOption:=0);
ETHERNET_CHASSIS_PLC_WARNING_DIFF(LIST:=LIST,Bit_Input:=GVL_Alarms.ETHERNET_CHASSIS_PLC_WARNING_DIFF,ID:=1104,Add_Info:='',Group:=App_Error_Group,HushOption:=0);
ETHERNET_CHASSIS_PLC_WARNING_FROZEN(LIST:=LIST,Bit_Input:=GVL_Alarms.ETHERNET_CHASSIS_PLC_WARNING_FROZEN,ID:=1105,Add_Info:='',Group:=App_Error_Group,HushOption:=0);

// Alarms_Monitor_App_STL_Body_CODE_GEN_STOP

END_PROGRAM

// Device/Application/LIBS/Alarms/Functions/Alarm_Log_Count_Errors
FUNCTION Alarm_Log_Count_Errors : INT

VAR_INPUT
	LIST: REFERENCE TO SLL_LOGGER_MAIN_SRUCT;
END_VAR
VAR_OUTPUT
END_VAR
VAR
	ErrorApp_Count:INT:=0;
	ErrorIO_Count:INT:=0;
	
	X:WORD;
END_VAR

ErrorApp_Count:=0;
ErrorIO_Count:=0;

FOR X :=0 TO (LIST.LOGGER_LIST_SIZE-1) BY 1 DO
	IF LIST.LOGGER_LIST[X].Group.ErrorApp THEN
		ErrorApp_Count:=ErrorApp_Count+1;		
	END_IF
	IF LIST.LOGGER_LIST[X].Group.ErrorIO THEN
		ErrorIO_Count:=ErrorIO_Count+1;
	END_IF
END_FOR

Alarm_Log_Count_Errors:=ErrorApp_Count+ErrorIO_Count;

END_FUNCTION

// Device/Application/LIBS/Alarms/Functions/Alarm_Log_Count_Warnings
FUNCTION Alarm_Log_Count_Warnings : INT

VAR_INPUT
	LIST: REFERENCE TO SLL_LOGGER_MAIN_SRUCT;
END_VAR
VAR_OUTPUT
END_VAR
VAR
	X:WORD;
	WarningsApp_Count:INT:=0;
	WarningsIO_Count:INT:=0;	
END_VAR

WarningsApp_Count:=0;
WarningsIO_Count:=0;

FOR X :=0 TO (LIST.LOGGER_LIST_SIZE-1) BY 1 DO
	IF LIST.LOGGER_LIST[X].Group.WarningApp THEN
		WarningsApp_Count:=WarningsApp_Count+1;
	END_IF
	IF LIST.LOGGER_LIST[X].Group.WarningIO THEN
		WarningsIO_Count:=WarningsIO_Count+1;
	END_IF
END_FOR
Alarm_Log_Count_Warnings:=WarningsApp_Count+WarningsIO_Count;

END_FUNCTION

// Device/Application/App_Common/VIZ/Viz_Common
PROGRAM Viz_Common
VAR_INPUT
END_VAR
VAR_OUTPUT
END_VAR
VAR
	INPUT_FAULT_FLASH_FAST_COUNT: INT;
	INPUT_FAULT_FLASH_SLOW_COUNT: INT;
	INIT: BOOL:=TRUE;
END_VAR
VAR // added by the converter: edge detectors and wires of the graphical bodies
    _w1, _w2 : BOOL;
END_VAR

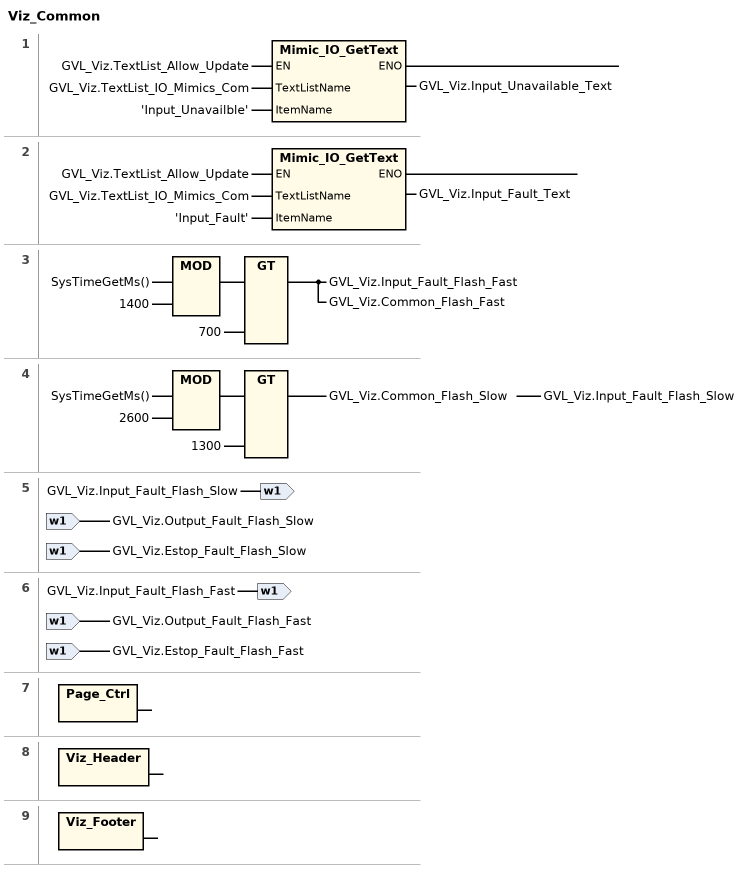
// NETWORK 1
IF GVL_Viz.TextList_Allow_Update THEN
    GVL_Viz.Input_Unavailable_Text := Mimic_IO_GetText(TextListName := GVL_Viz.TextList_IO_Mimics_Com, ItemName := 'Input_Unavailble');
END_IF

// NETWORK 2
IF GVL_Viz.TextList_Allow_Update THEN
    GVL_Viz.Input_Fault_Text := Mimic_IO_GetText(TextListName := GVL_Viz.TextList_IO_Mimics_Com, ItemName := 'Input_Fault');
END_IF

// NETWORK 3
_w1 := (SysTimeGetMs()) MOD 1400 > 700;
GVL_Viz.Input_Fault_Flash_Fast := _w1;
GVL_Viz.Common_Flash_Fast := _w1;

// NETWORK 4
_w2 := (SysTimeGetMs()) MOD 2600 > 1300;
GVL_Viz.Common_Flash_Slow := _w2;
GVL_Viz.Input_Fault_Flash_Slow := _w2;

// NETWORK 5
GVL_Viz.Output_Fault_Flash_Slow := GVL_Viz.Input_Fault_Flash_Slow;
GVL_Viz.Estop_Fault_Flash_Slow := GVL_Viz.Input_Fault_Flash_Slow;

// NETWORK 6
GVL_Viz.Output_Fault_Flash_Fast := GVL_Viz.Input_Fault_Flash_Fast;
GVL_Viz.Estop_Fault_Flash_Fast := GVL_Viz.Input_Fault_Flash_Fast;

// NETWORK 7
Page_Ctrl();

// NETWORK 8
Viz_Header();

// NETWORK 9
Viz_Footer();

END_PROGRAM

// Device/Application/LIBS/Mimic_IO_GetText
FUNCTION Mimic_IO_GetText : STRING
VAR_INPUT
	TextListName: STRING;
	ItemName:STRING;	
END_VAR
VAR
	Current : STRING:='';
	TextListItem:STRING:='';
END_VAR

Current := DynamicTextGetCurrentLanguage();

IF Current = '' THEN
	TextListItem:=DynamicTextGetDefaultText(ADR(TextListName), ADR(ItemName))^;
ELSE
	TextListItem:=DynamicTextGetText(ADR(TextListName), ADR(ItemName))^;
END_IF

// nothing found - just use the input!
IF TextListItem = '' THEN
	TextListItem:=ItemName;
END_IF

Mimic_IO_GetText:=TextListItem;

END_FUNCTION

// Device/Application/App_Common/Nav/Page Control/Page_Ctrl
PROGRAM Page_Ctrl
VAR
	HideManualIcon: BOOL;


	DrumArrow: RotatingArrow;
	
	Standard_CollectionArrow: MoveArrow_Angle;
	Standard_SideConvArrow: MoveArrow_Angle;
	Standard_TailConvArrow: MoveArrow_Angle;
	Standard_SideTransferArrow: MoveArrow_Angle;
	Standard_FeederArrow: MoveArrow_Angle;	
	
	Radial_StockpileArrow: MoveArrow_Angle;
	Radial_CollectionArrow_Ramp: MoveArrow_Angle;
	Radial_TailConveyor: MoveArrow_Angle;
	Radial_CollectionArrow_Flat: MoveArrow_Angle;
	Radial_Feeder: MoveArrow_Angle;
	
	StepMs: DWORD:=300;
END_VAR

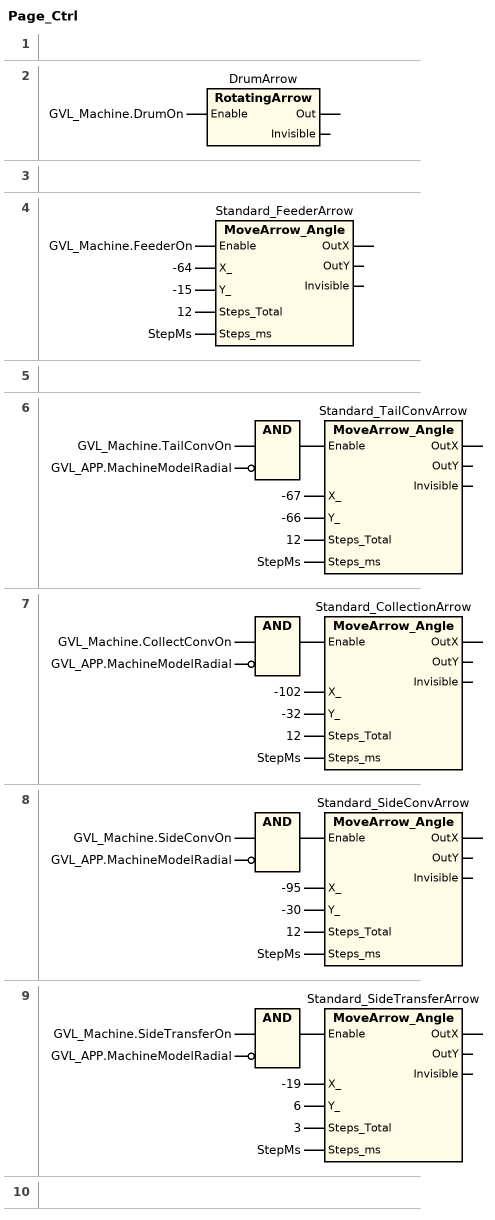
// NETWORK 1

// NETWORK 2
DrumArrow(Enable := GVL_Machine.DrumOn); // RotatingArrow

// NETWORK 3

// NETWORK 4
Standard_FeederArrow(
    Enable := GVL_Machine.FeederOn,
    X_ := -64,
    Y_ := -15,
    Steps_Total := 12,
    Steps_ms := StepMs); // MoveArrow_Angle

// NETWORK 5

// NETWORK 6
Standard_TailConvArrow(
    Enable := GVL_Machine.TailConvOn AND NOT GVL_APP.MachineModelRadial,
    X_ := -67,
    Y_ := -66,
    Steps_Total := 12,
    Steps_ms := StepMs); // MoveArrow_Angle

// NETWORK 7
Standard_CollectionArrow(
    Enable := GVL_Machine.CollectConvOn AND NOT GVL_APP.MachineModelRadial,
    X_ := -102,
    Y_ := -32,
    Steps_Total := 12,
    Steps_ms := StepMs); // MoveArrow_Angle

// NETWORK 8
Standard_SideConvArrow(
    Enable := GVL_Machine.SideConvOn AND NOT GVL_APP.MachineModelRadial,
    X_ := -95,
    Y_ := -30,
    Steps_Total := 12,
    Steps_ms := StepMs); // MoveArrow_Angle

// NETWORK 9
Standard_SideTransferArrow(
    Enable := GVL_Machine.SideTransferOn AND NOT GVL_APP.MachineModelRadial,
    X_ := -19,
    Y_ := 6,
    Steps_Total := 3,
    Steps_ms := StepMs); // MoveArrow_Angle

// NETWORK 10

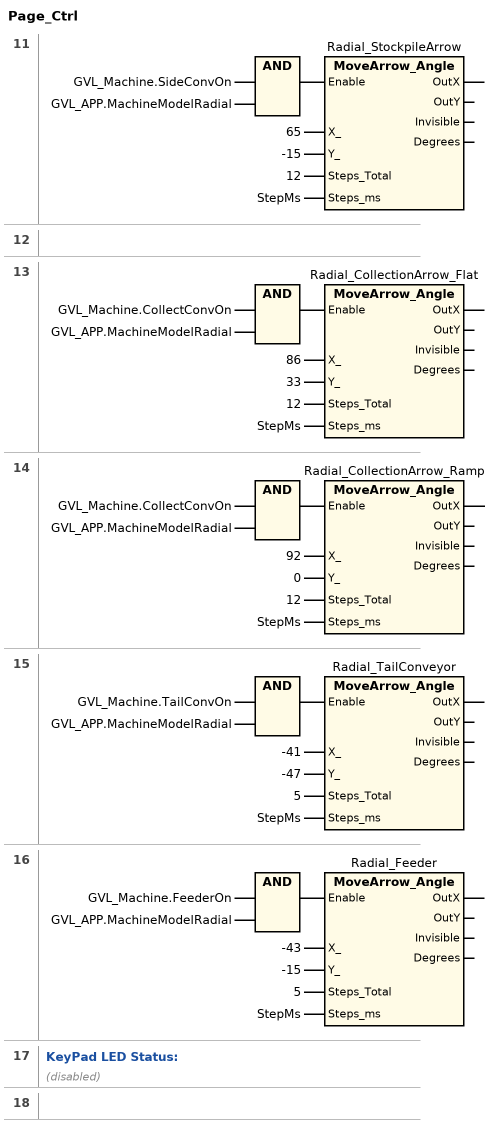
// NETWORK 11
Radial_StockpileArrow(
    Enable := GVL_Machine.SideConvOn AND GVL_APP.MachineModelRadial,
    X_ := 65,
    Y_ := -15,
    Steps_Total := 12,
    Steps_ms := StepMs); // MoveArrow_Angle

// NETWORK 12

// NETWORK 13
Radial_CollectionArrow_Flat(
    Enable := GVL_Machine.CollectConvOn AND GVL_APP.MachineModelRadial,
    X_ := 86,
    Y_ := 33,
    Steps_Total := 12,
    Steps_ms := StepMs); // MoveArrow_Angle

// NETWORK 14
Radial_CollectionArrow_Ramp(
    Enable := GVL_Machine.CollectConvOn AND GVL_APP.MachineModelRadial,
    X_ := 92,
    Y_ := 0,
    Steps_Total := 12,
    Steps_ms := StepMs); // MoveArrow_Angle

// NETWORK 15
Radial_TailConveyor(
    Enable := GVL_Machine.TailConvOn AND GVL_APP.MachineModelRadial,
    X_ := -41,
    Y_ := -47,
    Steps_Total := 5,
    Steps_ms := StepMs); // MoveArrow_Angle

// NETWORK 16
Radial_Feeder(
    Enable := GVL_Machine.FeederOn AND GVL_APP.MachineModelRadial,
    X_ := -43,
    Y_ := -15,
    Steps_Total := 5,
    Steps_ms := StepMs); // MoveArrow_Angle

// NETWORK 17 (disabled)
// label: KeyPad LED Status

// NETWORK 18

END_PROGRAM

// Device/Application/App_Common/Nav/Page Control/RotatingArrow
FUNCTION_BLOCK RotatingArrow
VAR_INPUT
	Enable: BOOL;
END_VAR
VAR_OUTPUT
	Out: INT;
	Invisible: BOOL;
END_VAR
VAR
	Ton1: TON;
	DegreeCount: INT;
END_VAR

Ton1(IN:= Enable AND NOT Ton1.Q, PT:=T#100MS);
IF Ton1.Q THEN
	DegreeCount:= DegreeCount + 10;
END_IF
IF DegreeCount>359 THEN DegreeCount:=0; END_IF
Out:=DegreeCount;
Invisible:= NOT Enable;

END_FUNCTION_BLOCK

// Device/Application/App_Common/Nav/Page Control/MoveArrow_Angle
FUNCTION_BLOCK MoveArrow_Angle
VAR_INPUT
	Enable: BOOL;
	X_:INT;
	Y_:INT;
	Steps_Total:DWORD;
	Steps_ms: DWORD;	
END_VAR
VAR_OUTPUT
	OutX: INT;
	OutY: INT;
	Invisible: BOOL;
END_VAR
VAR
	MillisStart:DWORD;
	MillisNext:DWORD;
	SkipCounter: DWORD;
	Step_index:DWORD;
	dwTimeRatio: DWORD;
END_VAR

IF Enable = 0 THEN
	Step_index := 0;
	MillisStart := 0;
	MillisNext:=0;
	Invisible:=TRUE;
	RETURN;
END_IF

IF MillisStart = 0 THEN
	// just started
	Invisible:=FALSE;
	MillisStart := SysTimeGetMs();
END_IF

IF MillisNext > 0  THEN
	IF SysTimeGetMs() < MillisNext THEN
		SkipCounter:=SkipCounter+1;
		RETURN; // nothing to do 
	END_IF
END_IF;

IF Step_index >= (Steps_Total-1) THEN
	MillisStart := SysTimeGetMs();
	Step_index:=0;
ELSE
	Step_index:=Step_index+1;
END_IF

MillisNext := MillisStart+(Steps_ms*Step_index);
dwTimeRatio :=  (Step_index*1000);
dwTimeRatio :=  dwTimeRatio/Steps_Total;

OutX := (X_ * TO_INT(dwTimeRatio))/1000;
OutY := (Y_ * TO_INT(dwTimeRatio))/1000;

END_FUNCTION_BLOCK

// Device/Application/App_Common/VIZ/Viz_Header
PROGRAM Viz_Header
VAR
	Battery_Warn_DUTY_CYCLE: DUTY_CYCLE;
	Header_Battery_Message: STRING;
	Header_Message_Show_Flash:BOOL;		
	Header_Message_DUTY_CYCLE: DUTY_CYCLE;
END_VAR

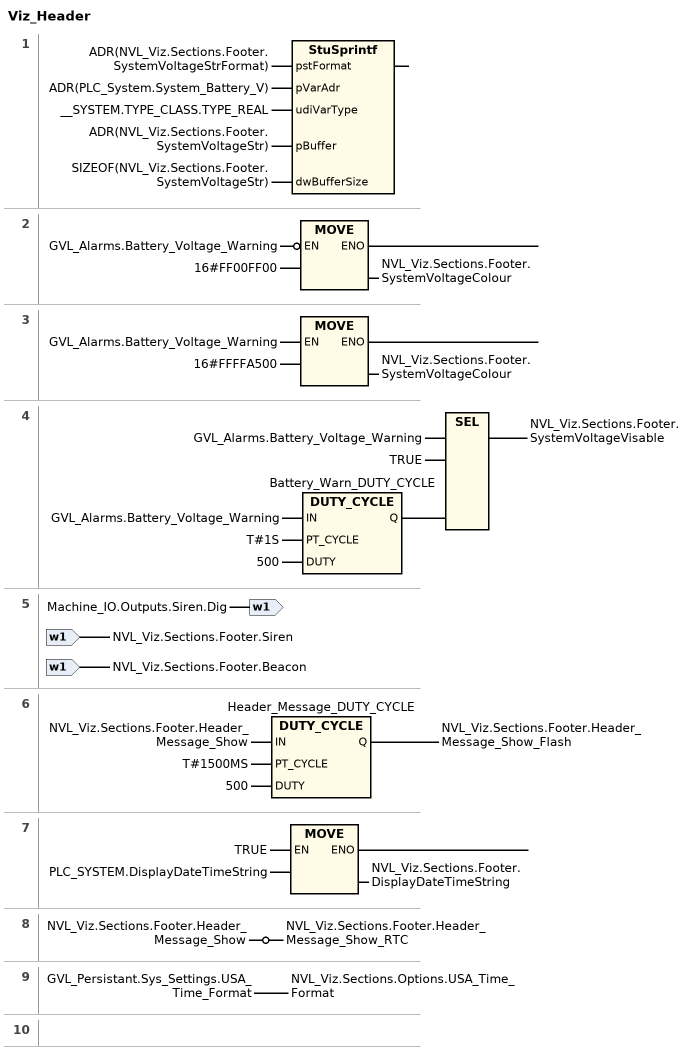
// NETWORK 1
StuSprintf(pstFormat := ADR(NVL_Viz.Sections.Footer.SystemVoltageStrFormat), pVarAdr := ADR(PLC_System.System_Battery_V), udiVarType := __SYSTEM.TYPE_CLASS.TYPE_REAL, pBuffer := ADR(NVL_Viz.Sections.Footer.SystemVoltageStr), dwBufferSize := SIZEOF(NVL_Viz.Sections.Footer.SystemVoltageStr));

// NETWORK 2
IF NOT GVL_Alarms.Battery_Voltage_Warning THEN NVL_Viz.Sections.Footer.SystemVoltageColour := 16#FF00FF00; END_IF

// NETWORK 3
IF GVL_Alarms.Battery_Voltage_Warning THEN NVL_Viz.Sections.Footer.SystemVoltageColour := 16#FFFFA500; END_IF

// NETWORK 4
Battery_Warn_DUTY_CYCLE(IN := GVL_Alarms.Battery_Voltage_Warning, PT_CYCLE := T#1S, DUTY := 500); // DUTY_CYCLE
NVL_Viz.Sections.Footer.SystemVoltageVisable := SEL(GVL_Alarms.Battery_Voltage_Warning, TRUE, Battery_Warn_DUTY_CYCLE.Q);

// NETWORK 5
NVL_Viz.Sections.Footer.Siren := Machine_IO.Outputs.Siren.Dig;
NVL_Viz.Sections.Footer.Beacon := Machine_IO.Outputs.Siren.Dig;

// NETWORK 6
Header_Message_DUTY_CYCLE(
    IN := NVL_Viz.Sections.Footer.Header_Message_Show,
    PT_CYCLE := T#1500MS,
    DUTY := 500); // DUTY_CYCLE
NVL_Viz.Sections.Footer.Header_Message_Show_Flash := Header_Message_DUTY_CYCLE.Q;

// NETWORK 7
NVL_Viz.Sections.Footer.DisplayDateTimeString := PLC_SYSTEM.DisplayDateTimeString;

// NETWORK 8
NVL_Viz.Sections.Footer.Header_Message_Show_RTC := NOT NVL_Viz.Sections.Footer.Header_Message_Show;

// NETWORK 9
NVL_Viz.Sections.Options.USA_Time_Format := GVL_Persistant.Sys_Settings.USA_Time_Format;

// NETWORK 10

END_PROGRAM

// Device/Application/App_Common/VIZ/Viz_Footer
PROGRAM Viz_Footer
VAR
	Footer_ShowDiagSwitch:BOOL;
	Footer_ShowAlmAck: BOOL;
	Footer_ShowNavLeft:BOOL;
	Footer_ShowNavRight:BOOL;
	Footer_ShowCAS:BOOL;	
END_VAR

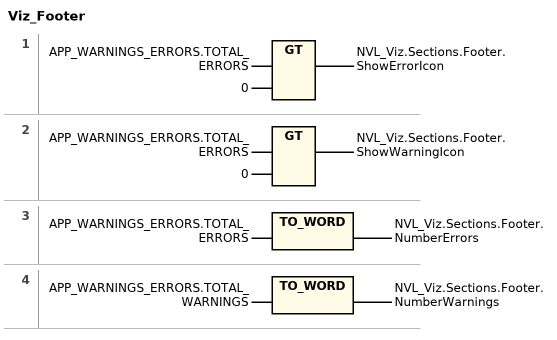
// NETWORK 1
NVL_Viz.Sections.Footer.ShowErrorIcon := APP_WARNINGS_ERRORS.TOTAL_ERRORS > 0;

// NETWORK 2
NVL_Viz.Sections.Footer.ShowWarningIcon := APP_WARNINGS_ERRORS.TOTAL_ERRORS > 0;

// NETWORK 3
NVL_Viz.Sections.Footer.NumberErrors := TO_WORD(APP_WARNINGS_ERRORS.TOTAL_ERRORS);

// NETWORK 4
NVL_Viz.Sections.Footer.NumberWarnings := TO_WORD(APP_WARNINGS_ERRORS.TOTAL_WARNINGS);

END_PROGRAM

// Device/Application/App_Common/UDP/UDP_COMS_TX
PROGRAM UDP_COMS_TX
VAR
		CYCLE_FREQ_FB_0: SLL_Common.CYCLE_FREQ;
END_VAR

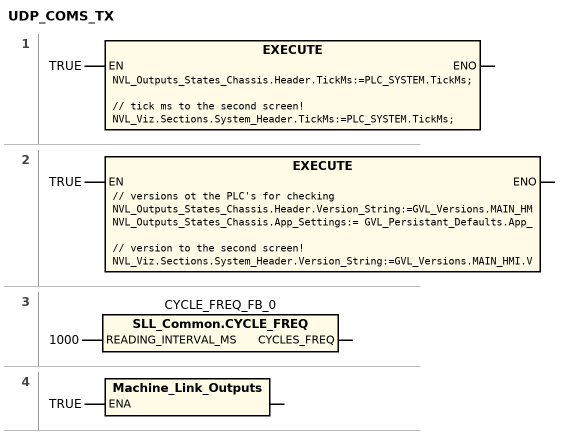
// NETWORK 1
NVL_Outputs_States_Chassis.Header.TickMs:=PLC_SYSTEM.TickMs;

// tick ms to the second screen!
NVL_Viz.Sections.System_Header.TickMs:=PLC_SYSTEM.TickMs;

// NETWORK 2
// versions ot the PLC's for checking
NVL_Outputs_States_Chassis.Header.Version_String:=GVL_Versions.MAIN_HMI.Version;
NVL_Outputs_States_Chassis.App_Settings:= GVL_Persistant_Defaults.App_Settings;

// version to the second screen!
NVL_Viz.Sections.System_Header.Version_String:=GVL_Versions.MAIN_HMI.Version;

// NETWORK 3
CYCLE_FREQ_FB_0(READING_INTERVAL_MS := 1000); // SLL_Common.CYCLE_FREQ

// NETWORK 4
Machine_Link_Outputs(ENA := TRUE);

END_PROGRAM

// Device/Application/App_CODE_GEN/MAIN_CODE_GEN/App_CODE_GEN/Machine IO/Funcs/Machine_Link_Outputs
PROGRAM Machine_Link_Outputs
VAR_INPUT
	ENA:BOOL;
END_VAR
VAR
	Init_Output_Links: BOOL := TRUE;
END_VAR

IF ENA = FALSE THEN
	RETURN;
END_IF

IF Init_Output_Links THEN
	Machine_Link_Outputs_Init();
	Init_Output_Links:=FALSE;
END_IF

// Machine_Link_Outputs_Main_CODE_GEN_START

// generated (UTC): 2024-07-23 18:31:25.127390+00:00
Machine_IO.Outputs.TAILCONVSPD_MA(); // CR0709.OUT0000
Machine_IO.Outputs.RHS_JACKLEGLOWER_OP(); // CR0709.OUT0001
Machine_IO.Outputs.SIDECONVSPD_MA(); // CR0709.OUT0002
Machine_IO.Outputs.LHS_JACKLEGRAISE_OP(); // CR0709.OUT0003
Machine_IO.Outputs.SIDETRANSFERSPD_MA(); // CR0709.OUT0004
Machine_IO.Outputs.LHS_JACKLEGLOWER_OP(); // CR0709.OUT0005
Machine_IO.Outputs.SETUPDUMPVALVE_OP(); // CR0709.OUT0006
Machine_IO.Outputs.COLLECTIONCONVSPD_MA(); // CR0709.OUT0007
Machine_IO.Outputs.COLLECTIONCONVON_OP(); // CR0709.OUT0008
Machine_IO.Outputs.SUPPLY_GROUP0(); // CR0709.GROUP0
Machine_IO.Outputs.DRUMSPD_MA_RAMP_LIMIT(); // CR0709.OUT0100
Machine_IO.Outputs.TRACKINGMODE(); // CR0709.OUT0101
Machine_IO.Outputs.FEEDERSPD_MA(); // CR0709.OUT0102
Machine_IO.Outputs.CRANKENABLE(); // CR0709.OUT0103
Machine_IO.Outputs.DIVERTOILTOTRACK_OP(); // CR0709.OUT0104
Machine_IO.Outputs.RHS_JACKLEGRAISE_OP(); // CR0709.OUT0105
Machine_IO.Outputs.TAILCONVON_OP(); // CR0709.OUT0106
Machine_IO.Outputs.SIDECONVON_OP(); // CR0709.OUT0107
Machine_IO.Outputs.SIDETRANSFERON_OP(); // CR0709.OUT0108
Machine_IO.Outputs.SUPPLY_GROUP1(); // CR0709.GROUP1
Machine_IO.Outputs.LEFTTRACKDIVERT_OP(); // CR0709.OUT0200
Machine_IO.Outputs.LTF_OP(); // CR0709.OUT0201
Machine_IO.Outputs.LTR_OP(); // CR0709.OUT0202
Machine_IO.Outputs.RIGHTTRACKDIVERT_OP(); // CR0709.OUT0203
Machine_IO.Outputs.RTF_OP(); // CR0709.OUT0204
Machine_IO.Outputs.RTR_OP(); // CR0709.OUT0205
Machine_IO.Outputs.DRUMONOFF_OP(); // CR0709.OUT0206
Machine_IO.Outputs.FEEDERONOFF_OP(); // CR0709.OUT0207
Machine_IO.Outputs.ECUENABLE(); // CR0709.OUT0208
Machine_IO.Outputs.SUPPLY_GROUP2(); // CR0709.GROUP2
Machine_IO.Outputs.SPARE_OUT3000(); // CR0709.OUT3000
Machine_IO.Outputs.SPARE_OUT3001(); // CR0709.OUT3001

// Machine_Link_Outputs_Main_CODE_GEN_STOP

Machine_IO.Outputs.Siren();
Machine_IO.Outputs.AUX_OP1();
Machine_IO.Outputs.AUX_OP2();

Machine_IO.Outputs.Siren();
Machine_IO.Outputs.AUX_OP1();
Machine_IO.Outputs.AUX_OP2();
Machine_IO.Outputs.FanFwd_OP();
Machine_IO.Outputs.FanRev_OP();
Machine_IO.Outputs.SideConvRaise_RadialLeft_OP();
Machine_IO.Outputs.SideConvLower_RadialRight_OP();
Machine_IO.Outputs.DivertValve();

END_PROGRAM

// Device/Application/App_CODE_GEN/MAIN_CODE_GEN/App_CODE_GEN/Machine IO/Funcs/Machine_Link_Outputs_Init
PROGRAM Machine_Link_Outputs_Init
VAR
END_VAR


// Machine_Link_Outputs_Init_CODE_GEN_START

// generated (UTC): 2024-07-23 18:31:25.139390+00:00

Machine_IO.Outputs.TAILCONVSPD_MA.Init('CHASSIS','TAILCONVSPD_MA','OUT0000','a16',NVL_Outputs_States_CHASSIS.All.OUT0000,NVL_IO_CHASSIS.All_Outputs_Diag.OUT0000,Machine_IO.Node_CHASSIS);
Machine_IO.Outputs.RHS_JACKLEGLOWER_OP.Init('CHASSIS','RHS_JACKLEGLOWER_OP','OUT0001','a17',NVL_Outputs_States_CHASSIS.All.OUT0001,NVL_IO_CHASSIS.All_Outputs_Diag.OUT0001,Machine_IO.Node_CHASSIS);
Machine_IO.Outputs.SIDECONVSPD_MA.Init('CHASSIS','SIDECONVSPD_MA','OUT0002','a18',NVL_Outputs_States_CHASSIS.All.OUT0002,NVL_IO_CHASSIS.All_Outputs_Diag.OUT0002,Machine_IO.Node_CHASSIS);
Machine_IO.Outputs.LHS_JACKLEGRAISE_OP.Init('CHASSIS','LHS_JACKLEGRAISE_OP','OUT0003','a19',NVL_Outputs_States_CHASSIS.All.OUT0003,NVL_IO_CHASSIS.All_Outputs_Diag.OUT0003,Machine_IO.Node_CHASSIS);
Machine_IO.Outputs.SIDETRANSFERSPD_MA.Init('CHASSIS','SIDETRANSFERSPD_MA','OUT0004','a20',NVL_Outputs_States_CHASSIS.All.OUT0004,NVL_IO_CHASSIS.All_Outputs_Diag.OUT0004,Machine_IO.Node_CHASSIS);
Machine_IO.Outputs.LHS_JACKLEGLOWER_OP.Init('CHASSIS','LHS_JACKLEGLOWER_OP','OUT0005','a21',NVL_Outputs_States_CHASSIS.All.OUT0005,NVL_IO_CHASSIS.All_Outputs_Diag.OUT0005,Machine_IO.Node_CHASSIS);
Machine_IO.Outputs.SETUPDUMPVALVE_OP.Init('CHASSIS','SETUPDUMPVALVE_OP','OUT0006','a22',NVL_Outputs_States_CHASSIS.All.OUT0006,NVL_IO_CHASSIS.All_Outputs_Diag.OUT0006,Machine_IO.Node_CHASSIS);
Machine_IO.Outputs.COLLECTIONCONVSPD_MA.Init('CHASSIS','COLLECTIONCONVSPD_MA','OUT0007','a23',NVL_Outputs_States_CHASSIS.All.OUT0007,NVL_IO_CHASSIS.All_Outputs_Diag.OUT0007,Machine_IO.Node_CHASSIS);
Machine_IO.Outputs.COLLECTIONCONVON_OP.Init('CHASSIS','COLLECTIONCONVON_OP','OUT0008','a24',NVL_Outputs_States_CHASSIS.All.OUT0008,NVL_IO_CHASSIS.All_Outputs_Diag.OUT0008,Machine_IO.Node_CHASSIS);

Machine_IO.Outputs.DRUMSPD_MA_RAMP_LIMIT.Init('CHASSIS','DRUMSPD_MA_RAMP_LIMIT','OUT0100','a6',NVL_Outputs_States_CHASSIS.All.OUT0100,NVL_IO_CHASSIS.All_Outputs_Diag.OUT0100,Machine_IO.Node_CHASSIS);
Machine_IO.Outputs.TRACKINGMODE.Init('CHASSIS','TRACKINGMODE','OUT0101','a7',NVL_Outputs_States_CHASSIS.All.OUT0101,NVL_IO_CHASSIS.All_Outputs_Diag.OUT0101,Machine_IO.Node_CHASSIS);
Machine_IO.Outputs.FEEDERSPD_MA.Init('CHASSIS','FEEDERSPD_MA','OUT0102','a8',NVL_Outputs_States_CHASSIS.All.OUT0102,NVL_IO_CHASSIS.All_Outputs_Diag.OUT0102,Machine_IO.Node_CHASSIS);
Machine_IO.Outputs.CRANKENABLE.Init('CHASSIS','CRANKENABLE','OUT0103','a9',NVL_Outputs_States_CHASSIS.All.OUT0103,NVL_IO_CHASSIS.All_Outputs_Diag.OUT0103,Machine_IO.Node_CHASSIS);
Machine_IO.Outputs.DIVERTOILTOTRACK_OP.Init('CHASSIS','DIVERTOILTOTRACK_OP','OUT0104','a10',NVL_Outputs_States_CHASSIS.All.OUT0104,NVL_IO_CHASSIS.All_Outputs_Diag.OUT0104,Machine_IO.Node_CHASSIS);
Machine_IO.Outputs.RHS_JACKLEGRAISE_OP.Init('CHASSIS','RHS_JACKLEGRAISE_OP','OUT0105','a11',NVL_Outputs_States_CHASSIS.All.OUT0105,NVL_IO_CHASSIS.All_Outputs_Diag.OUT0105,Machine_IO.Node_CHASSIS);
Machine_IO.Outputs.TAILCONVON_OP.Init('CHASSIS','TAILCONVON_OP','OUT0106','a12',NVL_Outputs_States_CHASSIS.All.OUT0106,NVL_IO_CHASSIS.All_Outputs_Diag.OUT0106,Machine_IO.Node_CHASSIS);
Machine_IO.Outputs.SIDECONVON_OP.Init('CHASSIS','SIDECONVON_OP','OUT0107','a13',NVL_Outputs_States_CHASSIS.All.OUT0107,NVL_IO_CHASSIS.All_Outputs_Diag.OUT0107,Machine_IO.Node_CHASSIS);
Machine_IO.Outputs.SIDETRANSFERON_OP.Init('CHASSIS','SIDETRANSFERON_OP','OUT0108','a14',NVL_Outputs_States_CHASSIS.All.OUT0108,NVL_IO_CHASSIS.All_Outputs_Diag.OUT0108,Machine_IO.Node_CHASSIS);

Machine_IO.Outputs.LEFTTRACKDIVERT_OP.Init('CHASSIS','LEFTTRACKDIVERT_OP','OUT0200','a73',NVL_Outputs_States_CHASSIS.All.OUT0200,NVL_IO_CHASSIS.All_Outputs_Diag.OUT0200,Machine_IO.Node_CHASSIS);
Machine_IO.Outputs.LTF_OP.Init('CHASSIS','LTF_OP','OUT0201','a74',NVL_Outputs_States_CHASSIS.All.OUT0201,NVL_IO_CHASSIS.All_Outputs_Diag.OUT0201,Machine_IO.Node_CHASSIS);
Machine_IO.Outputs.LTR_OP.Init('CHASSIS','LTR_OP','OUT0202','a75',NVL_Outputs_States_CHASSIS.All.OUT0202,NVL_IO_CHASSIS.All_Outputs_Diag.OUT0202,Machine_IO.Node_CHASSIS);
Machine_IO.Outputs.RIGHTTRACKDIVERT_OP.Init('CHASSIS','RIGHTTRACKDIVERT_OP','OUT0203','a76',NVL_Outputs_States_CHASSIS.All.OUT0203,NVL_IO_CHASSIS.All_Outputs_Diag.OUT0203,Machine_IO.Node_CHASSIS);
Machine_IO.Outputs.RTF_OP.Init('CHASSIS','RTF_OP','OUT0204','a77',NVL_Outputs_States_CHASSIS.All.OUT0204,NVL_IO_CHASSIS.All_Outputs_Diag.OUT0204,Machine_IO.Node_CHASSIS);
Machine_IO.Outputs.RTR_OP.Init('CHASSIS','RTR_OP','OUT0205','a78',NVL_Outputs_States_CHASSIS.All.OUT0205,NVL_IO_CHASSIS.All_Outputs_Diag.OUT0205,Machine_IO.Node_CHASSIS);
Machine_IO.Outputs.DRUMONOFF_OP.Init('CHASSIS','DRUMONOFF_OP','OUT0206','a79',NVL_Outputs_States_CHASSIS.All.OUT0206,NVL_IO_CHASSIS.All_Outputs_Diag.OUT0206,Machine_IO.Node_CHASSIS);
Machine_IO.Outputs.FEEDERONOFF_OP.Init('CHASSIS','FEEDERONOFF_OP','OUT0207','a80',NVL_Outputs_States_CHASSIS.All.OUT0207,NVL_IO_CHASSIS.All_Outputs_Diag.OUT0207,Machine_IO.Node_CHASSIS);
Machine_IO.Outputs.ECUENABLE.Init('CHASSIS','ECUENABLE','OUT0208','a81',NVL_Outputs_States_CHASSIS.All.OUT0208,NVL_IO_CHASSIS.All_Outputs_Diag.OUT0208,Machine_IO.Node_CHASSIS);

Machine_IO.Outputs.SPARE_OUT3000.Init('CHASSIS','SPARE_OUT3000','OUT3000','a31',NVL_Outputs_States_CHASSIS.All.OUT3000,NVL_IO_CHASSIS.All_Outputs_Diag.OUT3000,Machine_IO.Node_CHASSIS);
Machine_IO.Outputs.SPARE_OUT3001.Init('CHASSIS','SPARE_OUT3001','OUT3001','a32',NVL_Outputs_States_CHASSIS.All.OUT3001,NVL_IO_CHASSIS.All_Outputs_Diag.OUT3001,Machine_IO.Node_CHASSIS);

Machine_IO.Outputs.SUPPLY_GROUP0.Init('CHASSIS','SUPPLY_GROUP0','GROUP0','a1',NVL_Outputs_States_CHASSIS.All.GROUP0,NVL_IO_CHASSIS.All_Outputs_Diag.GROUP0,Machine_IO.Node_CHASSIS);
Machine_IO.Outputs.SUPPLY_GROUP1.Init('CHASSIS','SUPPLY_GROUP1','GROUP0','a1',NVL_Outputs_States_CHASSIS.All.GROUP1,NVL_IO_CHASSIS.All_Outputs_Diag.GROUP1,Machine_IO.Node_CHASSIS);
Machine_IO.Outputs.SUPPLY_GROUP2.Init('CHASSIS','SUPPLY_GROUP2','GROUP0','a1',NVL_Outputs_States_CHASSIS.All.GROUP2,NVL_IO_CHASSIS.All_Outputs_Diag.GROUP2,Machine_IO.Node_CHASSIS);

// Machine_Link_Outputs_Init_CODE_GEN_STOP

Machine_IO.Outputs.SIREN.Init('AUX','SIREN_BEACON','OP0','',GVL_CAN_TX_AUX.OUTPUTS.OP0,Machine_IO.Node_AUX);
Machine_IO.Outputs.AUX_OP1.Init('AUX','SPARE_OP1','OP1','',GVL_CAN_TX_AUX.OUTPUTS.OP1,Machine_IO.Node_AUX);
Machine_IO.Outputs.AUX_OP2.Init('AUX','SPARE_OP2','OP2','',GVL_CAN_TX_AUX.OUTPUTS.OP2,Machine_IO.Node_AUX);
Machine_IO.Outputs.DivertValve.Init('AUX','DIVERT_VALVE','OP3','',GVL_CAN_TX_AUX.OUTPUTS.OP3,Machine_IO.Node_AUX);
Machine_IO.Outputs.FanFwd_OP.Init('AUX','FAN_FORWARD','OP4','',GVL_CAN_TX_AUX.OUTPUTS.OP4,Machine_IO.Node_AUX);
Machine_IO.Outputs.FanRev_OP.Init('AUX','FAN_REVERSE','OP5','',GVL_CAN_TX_AUX.OUTPUTS.OP5,Machine_IO.Node_AUX);
Machine_IO.Outputs.SideConvRaise_RadialLeft_OP.Init('AUX','SIDE_CONV_RAISE/RADIAL_LEFT','OP6','',GVL_CAN_TX_AUX.OUTPUTS.OP6,Machine_IO.Node_AUX);
Machine_IO.Outputs.SideConvLower_RadialRight_OP.Init('AUX','SIDE_CONV_LOWER/RADIAL_RIGHT','OP7','',GVL_CAN_TX_AUX.OUTPUTS.OP7,Machine_IO.Node_AUX);

END_PROGRAM

// Device/Application/LIBS/IO Diagnostics/CRXXXX_Input_Display
FUNCTION_BLOCK CRXXXX_Input_Display
VAR_INPUT

END_VAR
VAR_OUTPUT
	oPinDetailsStr:STRING;
	oSignalNameStr: STRING;
	oMainString: STRING; // could be Digital:ON/OFF, mV, mA or Hz?
	oMainStringColour:DWORD;
	oDiagStr: STRING; // Diagnostics info
	oShowDigRect:BOOL;
	oDigRectColour:DWORD;
	oTypeStr:STRING;
END_VAR
VAR
	InitDone:BOOL :=FALSE;
	IpREF: REFERENCE TO IpCom;
	
	Update: BOOL:=TRUE;
	Update_Signal_Name: BOOL:=TRUE;
	
	temp_real:STRING(10);
	TextListItem:STRING;	

	UpdateDiag: BOOL:=FALSE;
	MainStringFlash: BOOL;
	MainStringTemp: STRING;
END_VAR

IF Update=FALSE THEN
	RETURN;
END_IF

IF __ISVALIDREF(IpREF) = FALSE THEN
	RETURN;
END_IF

IF IpREF.RefsOK = FALSE THEN
	RETURN;
END_IF

// this code displays the Signal name - can be toggled using the function key
IF Update_Signal_Name THEN
	//oPinDetailsStr:=IpREF.Pin_Details;	
	oPinDetailsStr:=IpREF.Pin_Name;	
	IF GVL_Viz.Diag_Signal_Name_Toggle THEN
		TextListItem:=IpREF.Signal_Name;
	ELSE
		TextListItem:=Mimic_IO_GetText(GVL_Viz.TextList_IO_Diag,IpREF.PLC_IO_Ref);
	END_IF	
	
	IF (FIND(TextListItem,'Spare_') = 1) OR (FIND(TextListItem,'SPARE_') = 1) THEN
		// Starts with Spare
		oSignalNameStr:=' --- ';
	ELSE
		oSignalNameStr:=TextListItem;
	END_IF
END_IF

// set defaults first for the main string
oMainString:='';
MainStringTemp:='';
MainStringFlash:=FALSE;
oMainStringColour:=GVL_Viz.Diag_Input_Font_Colour_OK;

IF IpREF.Unavail THEN
	IF GVL_Viz.Input_Fault_Flash_Slow THEN
		oMainString:=GVL_Viz.Diag_Input_Unavailable_Text;
		MainStringFlash:=TRUE;	
	END_IF
	oMainStringColour:=GVL_Viz.Diag_Input_Font_Colour_Unavail;
END_IF

IF IpREF.Fault THEN
	IF GVL_Viz.Input_Fault_Flash_Slow THEN
		MainStringFlash:=TRUE;
		oMainString:=GVL_Viz.Diag_Input_Pin_Fault_Text;
	END_IF
	oMainStringColour:=GVL_Viz.Diag_Input_Font_Colour_Fault;
END_IF

CASE IpREF.PLC_INPUT_DATA.eMode OF
ifmIOcommon.MODE_INPUT.IN_DIGITAL_CSI:
	oShowDigRect:=TRUE;
	oTypeStr:='CSI';
	
	temp_real:=OSCAT_BASIC.REAL_TO_STRF(TO_REAL(IpREF.PLC_INPUT_DATA.uiValueAnalogue)/1000,2,'.');
	MainStringTemp:=CONCAT(temp_real,'V');
	
	IF LEN(IpREF.DiagString) = 0 THEN
		IF IpREF.PLC_INPUT_DATA.xValueDigital = TRUE THEN
			oDigRectColour:=GVL_Viz.IFM_IO_Input_DigRectColour_ON;
			MainStringTemp:= CONCAT(MainStringTemp,', ON');
		ELSE
			oDigRectColour:=GVL_Viz.IFM_IO_Input_DigRectColour_OFF;		
			MainStringTemp:= CONCAT(MainStringTemp,', OFF');
		END_IF
		
		MainStringTemp:= CONCAT(MainStringTemp,',D:');
		MainStringTemp:= CONCAT(MainStringTemp,TO_STRING(IpREF.DeltaMs));
	
		MainStringTemp:= CONCAT(MainStringTemp,',C:');
		MainStringTemp:= CONCAT(MainStringTemp,TO_STRING(IpREF.PLC_INPUT_DATA.DigitalChanges));		
	ELSE
		UpdateDiag:=TRUE; // just use the diagnostic string!
	END_IF
	

ifmIOcommon.MODE_INPUT.IN_DIGITAL_CSO:
	oShowDigRect:=TRUE;
	oTypeStr:='CSO';
	
	temp_real:=OSCAT_BASIC.REAL_TO_STRF(TO_REAL(IpREF.PLC_INPUT_DATA.uiValueAnalogue)/1000,2,'.');
	MainStringTemp:=CONCAT(temp_real,'V');
	
	IF IpREF.PLC_INPUT_DATA.xValueDigital = TRUE THEN
		oDigRectColour:=GVL_Viz.IFM_IO_Input_DigRectColour_ON;
		MainStringTemp:= CONCAT(MainStringTemp,', ON');
	ELSE
		oDigRectColour:=GVL_Viz.IFM_IO_Input_DigRectColour_OFF;		
		MainStringTemp:= CONCAT(MainStringTemp,', OFF');
	END_IF

	MainStringTemp:= CONCAT(MainStringTemp,',D:');
	MainStringTemp:= CONCAT(MainStringTemp,TO_STRING(IpREF.DeltaMs));

	MainStringTemp:= CONCAT(MainStringTemp,',C:');
	MainStringTemp:= CONCAT(MainStringTemp,TO_STRING(IpREF.PLC_INPUT_DATA.DigitalChanges));
	
ifmIOcommon.MODE_INPUT.MONITOR:
	CASE IpREF.PLC_INPUT_DATA.Signal_Type OF
	Diag_Ip_Signal_Enum.FreqPulseHigh:
	 	oTypeStr:='FrqH';
	 	oShowDigRect:=FALSE;
	 	UpdateDiag:=TRUE;	
	Diag_Ip_Signal_Enum.FreqPulseLow:
	 	oTypeStr:='FrqL';
	 	oShowDigRect:=FALSE;
	 	UpdateDiag:=TRUE;		
	END_CASE
	
ifmIOcommon.MODE_INPUT.IN_CURRENT_CSI:
	oTypeStr:='4-20ma';
	oShowDigRect:=FALSE;
	MainStringTemp:= 'Raw:';
	temp_real:=OSCAT_BASIC.REAL_TO_STRF(TO_REAL(IpREF.PLC_INPUT_DATA.uiValueAnalogue)/1000,2,'.');
	MainStringTemp:= CONCAT(MainStringTemp,temp_real);
	MainStringTemp:= CONCAT(MainStringTemp,'ma');
	UpdateDiag:=TRUE;

ifmIOcommon.MODE_INPUT.IN_RESISTOR:
	oTypeStr:='Res';
	oShowDigRect:=FALSE;
	MainStringTemp:= 'Resistance:';
	MainStringTemp:= CONCAT(MainStringTemp,UINT_TO_STRING(IpREF.PLC_INPUT_DATA.uiValueAnalogue));
	MainStringTemp:= CONCAT(MainStringTemp,' Ohms');
	UpdateDiag:=TRUE;

ifmIOcommon.MODE_INPUT.IN_VOLTAGE_32:
	oTypeStr:='0-32v';
	oShowDigRect:=FALSE;
	MainStringTemp:= 'Raw:';
	MainStringTemp:= CONCAT(MainStringTemp,UINT_TO_STRING(IpREF.PLC_INPUT_DATA.uiValueAnalogue));
	MainStringTemp:= CONCAT(MainStringTemp,'mV');
	UpdateDiag:=TRUE;

ifmIOcommon.MODE_INPUT.IN_VOLTAGE_10:
	oTypeStr:='0-10v';
	oShowDigRect:=FALSE;
	MainStringTemp:= 'Raw:';
	MainStringTemp:= CONCAT(MainStringTemp,UINT_TO_STRING(IpREF.PLC_INPUT_DATA.uiValueAnalogue));
	MainStringTemp:= CONCAT(MainStringTemp,'mV');
	UpdateDiag:=TRUE;
	
ifmIOcommon.MODE_INPUT.UNCHANGED:
	UpdateDiag:=TRUE;	
END_CASE

IF 	UpdateDiag=TRUE THEN
	IF LEN(IpREF.DiagString) > 0 THEN
		IF LEN(MainStringTemp) > 0 THEN
			MainStringTemp:= CONCAT(MainStringTemp,',');		
		END_IF
		MainStringTemp:= CONCAT(MainStringTemp,IpREF.DiagString);
	END_IF	
END_IF

IF MainStringFlash = FALSE THEN
	oMainString:=MainStringTemp;
END_IF
oDiagStr:='Diag. OK';

METHOD Init : BOOL
VAR_INPUT
	pIpREF: REFERENCE TO IpCom;
END_VAR
IpREF REF= pIpREF;
InitDone:=TRUE;
END_METHOD

END_FUNCTION_BLOCK

// Device/Application/LIBS/IO Common/IpCom
FUNCTION_BLOCK PUBLIC IpCom

VAR_INPUT
	Dig: BOOL;
	uValue: WORD;
	
	DiagString: STRING:='';
	ScaledString: STRING:='';
	ScaledReal: REAL;	
END_VAR

VAR_OUTPUT	
END_VAR

VAR
	PLC_INPUT_DATA: REFERENCE TO CRXXXX_INPUT_DATA;
	PLC_Name: STRING;
	Signal_Name: STRING;
	Pin_Name: STRING;
	Pin_Details: STRING;
	
	NodeFB: REFERENCE TO NodeComFB;
	
	Unavail: BOOL;
	Fault: BOOL;
	
	RefsOK: BOOL;
	
	Diag_OK:BOOL;
	Diag_Error:BOOL;
	Diag_Warn:BOOL;
	Diag_Other:BOOL;	
		
	DigitalChangesPrev:WORD;
	
	DeltaMs: UDINT;
	ChangeMs: UDINT;
	
	DiagInfo:STRING:='';
	PLC_IO_Ref:STRING;
	
	Alarm_eDiagInfo:ifmTypes.DIAG_INFO;		
	AlmLog: IO_LogCom;
	Alarm_Active: BOOL;		
END_VAR

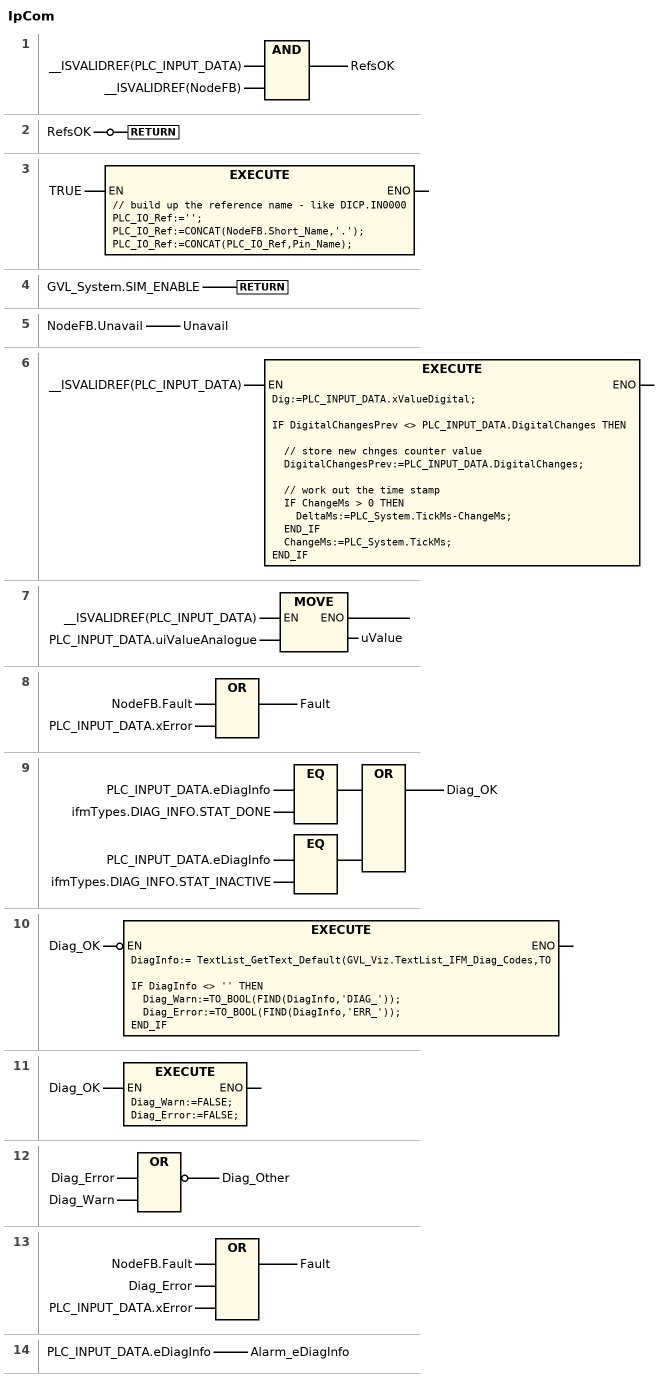
// NETWORK 1
RefsOK := (__ISVALIDREF(PLC_INPUT_DATA)) AND (__ISVALIDREF(NodeFB));

// NETWORK 2
IF NOT RefsOK THEN RETURN; END_IF

// NETWORK 3
// build up the reference name - like DICP.IN0000
PLC_IO_Ref:='';
PLC_IO_Ref:=CONCAT(NodeFB.Short_Name,'.');
PLC_IO_Ref:=CONCAT(PLC_IO_Ref,Pin_Name);

// NETWORK 4
IF GVL_System.SIM_ENABLE THEN RETURN; END_IF

// NETWORK 5
Unavail := NodeFB.Unavail;

// NETWORK 6
IF __ISVALIDREF(PLC_INPUT_DATA) THEN
    Dig:=PLC_INPUT_DATA.xValueDigital;
    
    IF DigitalChangesPrev <> PLC_INPUT_DATA.DigitalChanges THEN 
    
    	// store new chnges counter value
    	DigitalChangesPrev:=PLC_INPUT_DATA.DigitalChanges;
    
    	// work out the time stamp
    	IF ChangeMs > 0 THEN
    		DeltaMs:=PLC_System.TickMs-ChangeMs;
    	END_IF
    	ChangeMs:=PLC_System.TickMs;
    END_IF
END_IF

// NETWORK 7
IF __ISVALIDREF(PLC_INPUT_DATA) THEN uValue := PLC_INPUT_DATA.uiValueAnalogue; END_IF

// NETWORK 8
Fault := NodeFB.Fault OR PLC_INPUT_DATA.xError;

// NETWORK 9
Diag_OK := PLC_INPUT_DATA.eDiagInfo = ifmTypes.DIAG_INFO.STAT_DONE OR PLC_INPUT_DATA.eDiagInfo = ifmTypes.DIAG_INFO.STAT_INACTIVE;

// NETWORK 10
IF NOT Diag_OK THEN
    DiagInfo:= TextList_GetText_Default(GVL_Viz.TextList_IFM_Diag_Codes,TO_STRING(PLC_INPUT_DATA.eDiagInfo));
    
    IF DiagInfo <> '' THEN
    	Diag_Warn:=TO_BOOL(FIND(DiagInfo,'DIAG_'));	
    	Diag_Error:=TO_BOOL(FIND(DiagInfo,'ERR_'));	
    END_IF
END_IF

// NETWORK 11
IF Diag_OK THEN
    Diag_Warn:=FALSE;
    Diag_Error:=FALSE;
END_IF

// NETWORK 12
Diag_Other := NOT (Diag_Error OR Diag_Warn);

// NETWORK 13
Fault := NodeFB.Fault OR Diag_Error OR PLC_INPUT_DATA.xError;

// NETWORK 14
Alarm_eDiagInfo := PLC_INPUT_DATA.eDiagInfo;

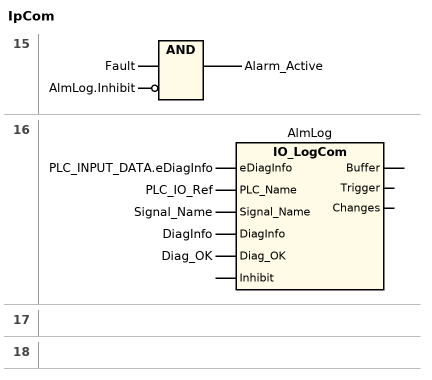
// NETWORK 15
Alarm_Active := Fault AND NOT AlmLog.Inhibit;

// NETWORK 16
AlmLog(
    eDiagInfo := PLC_INPUT_DATA.eDiagInfo,
    PLC_Name := PLC_IO_Ref,
    Signal_Name := Signal_Name,
    DiagInfo := DiagInfo,
    Diag_OK := Diag_OK); // IO_LogCom

// NETWORK 17

// NETWORK 18

METHOD Init : BOOL
VAR_INPUT
	pPLC_Name: STRING;
	pSignal_Name: STRING;
	pPin_Name: STRING;
	pPin_Details: STRING;
	pPLC_INPUT_DATA: REFERENCE TO CRXXXX_INPUT_DATA;
	pNodeFB: REFERENCE TO NodeComFB;
END_VAR
PLC_Name:=pPLC_Name;
Signal_Name:=pSignal_Name;
Pin_Name:=pPin_Name;
Pin_Details:=pPin_Details;

PLC_INPUT_DATA REF= pPLC_INPUT_DATA;

NodeFB REF=pNodeFB;
END_METHOD

END_FUNCTION_BLOCK

// Device/Application/LIBS/TextList_GetText_Default
FUNCTION TextList_GetText_Default : STRING
VAR_INPUT
	TextListName: STRING;
	ItemName:STRING;	
END_VAR
VAR
	TextListItemPtr:POINTER TO STRING;
	TextListItem:STRING:='';	
END_VAR

TextListItemPtr:=ADR(TextListItem);
TextListName:='TextList_IFM_Diag_Codes';
//TextListItemPtr:=DynamicTextGetDefaultTextW(ADR(TextListName), ADR(ItemName));
TextListItemPtr:=DynamicTextGetDefaultText(ADR(TextListName), ADR(ItemName));

TextList_GetText_Default:=TextListItem;

END_FUNCTION

// Device/Application/LIBS/IO Common/IO_LogCom
FUNCTION_BLOCK IO_LogCom
VAR_INPUT
	eDiagInfo: ifmTypes.DIAG_INFO;
	PLC_Name: REFERENCE TO STRING;
	Signal_Name: REFERENCE TO STRING;
	DiagInfo: REFERENCE TO STRING;
	Diag_OK: BOOL;
	Inhibit: BOOL:=FALSE;
END_VAR
VAR_OUTPUT
	Buffer:STRING;
	Trigger:BOOL:=FALSE;
	Changes:WORD:=0;
END_VAR
VAR
	Buffer_:STRING:='';
	eDiagInfo_prev: ifmTypes.DIAG_INFO;	
	Log_Change_Cycles:WORD:=0;
	Create_Alarm:BOOL;
	Create_Alarm_Count:WORD;
	TriggerTimestamp:UDINT;
	TriggerPulse_ms:UDINT;
	Diff:UDINT;
END_VAR
VAR_IN_OUT
END_VAR

Create_Alarm:=FALSE;

IF TriggerPulse_ms > 0 THEN
	// pulse active...
	IF (PLC_SYSTEM.TickMs - TriggerPulse_ms) > 100 THEN
		TriggerPulse_ms:=0;
		Trigger:=FALSE;
	END_IF
END_IF

IF eDiagInfo_prev <> eDiagInfo THEN
	// DiagInfo has changed...
	Changes:=Changes+1;
	TriggerTimestamp:=PLC_SYSTEM.TickMs;	
	eDiagInfo_prev:=eDiagInfo;
ELSE
	// DiagInfo is steady..
	IF TriggerTimestamp>0 THEN
		Diff := PLC_SYSTEM.TickMs - TriggerTimestamp; 
		IF Diff >= 100 THEN	
			IF Diag_OK = FALSE AND Inhibit = FALSE THEN
				TriggerTimestamp:=PLC_SYSTEM.TickMs;
				Create_Alarm:=TRUE;
			END_IF
		END_IF		
	END_IF
END_IF

IF Create_Alarm THEN
	// log string - can show more info!
	Buffer_:='';
	Buffer_:=CONCAT(Buffer_,PLC_Name);
	Buffer_:=CONCAT(Buffer_,'.');
	Buffer_:=CONCAT(Buffer_,Signal_Name);
	Buffer_:=CONCAT(Buffer_,':');
	Buffer_:=CONCAT(Buffer_,DiagInfo);	
	Log_File_Append(LogString:=Buffer_,szFileName:=GVL_Logging.Main_Log_Filename,GVL_Logging.Main_Log_Filename_Updated);
	
	// alarm buffer string - less is ok!
	Buffer_:='';
	Buffer_:=CONCAT(Buffer_,DiagInfo);
	
	Buffer:=TO_STRING(Buffer_);
	TriggerTimestamp:=0;
	Trigger:=TRUE;
	TriggerPulse_ms := PLC_SYSTEM.TickMs;
	Create_Alarm_Count:=Create_Alarm_Count+1;
END_IF

END_FUNCTION_BLOCK

// Device/Application/LIBS/IO Common/OpCom
FUNCTION_BLOCK OpCom

VAR_INPUT
//	Dig: BOOL;
	DiagString: STRING:='';
	Value: UINT;
END_VAR

VAR
	OUTPUT_STATE_DATA:  REFERENCE TO CRXXXX_OUTPUT_STATE_DATA;
	OUTPUT_DIAG_DATA: REFERENCE TO CRXXXX_OUTPUT_DATA;
	
	SET_UPDATES: DWORD;	
	PLC_Name: STRING;
	Signal_Name: STRING;
	Pin_Name: STRING;
	Pin_Details: STRING;
	
	NodeFB: REFERENCE TO NodeComFB;
	
	RefsOK: BOOL;
	
	Diag_OK:BOOL;
	Diag_Error:BOOL;
	Diag_Warn:BOOL;
	Diag_Other:BOOL;
	
	Fault:BOOL;	
	Unavail:BOOL;
	GroupSupplyOn:BOOL;
	
	DiagInfo:STRING:='';	
	PLC_IO_Ref:STRING;	
	
	Alarm_eDiagInfo:ifmTypes.DIAG_INFO;	
	AlmLog: IO_LogCom;
	Alarm_Active: BOOL;		
END_VAR

VAR_OUTPUT
	DigOn: BOOL;
END_VAR

